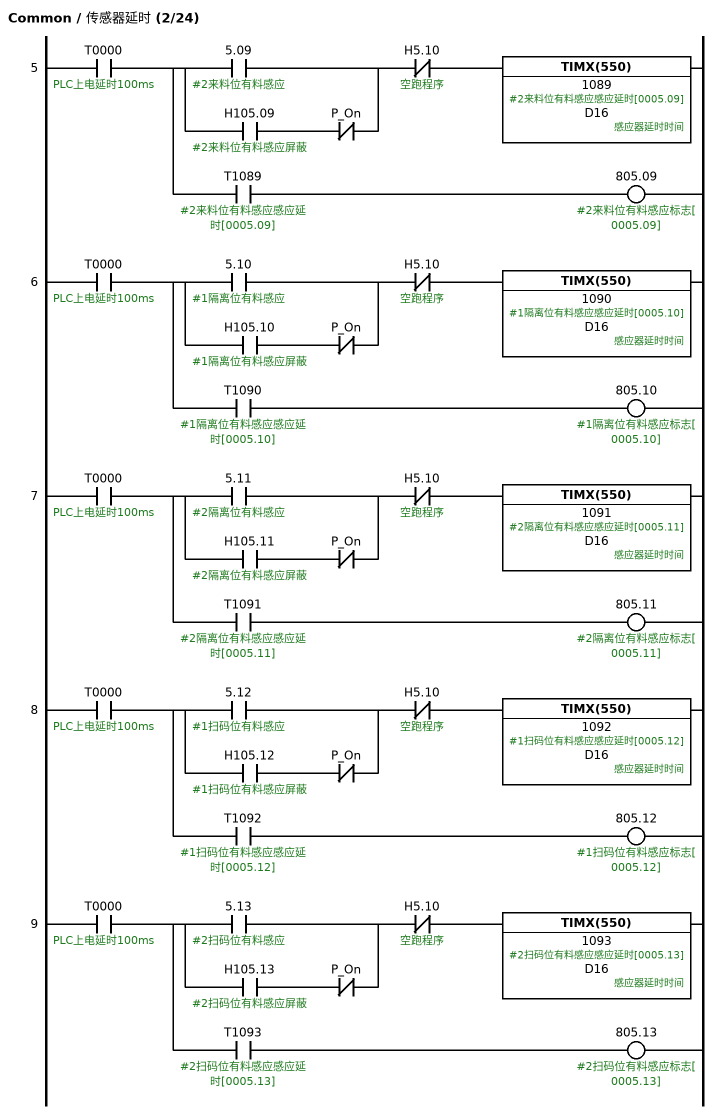
; [picture p504: Common / 传感器延时, rungs 5-9]
; rung 5
LD T0000  ; PLC上电延时100ms
OUT TR0
LD 5.09  ; #2来料位有料感应
LD H105.09  ; #2来料位有料感应屏蔽
ANDNOT P_On
ORLD
ANDLD
ANDNOT H5.10  ; 空跑程序
TIMX(550) 1089 D16  ; 感应器延时时间, #2来料位有料感应感应延时[0005.09]
LD TR0
AND T1089  ; #2来料位有料感应感应延时[0005.09]
OUT 805.09  ; #2来料位有料感应标志[0005.09]
; rung 6
LD T0000  ; PLC上电延时100ms
OUT TR0
LD 5.10  ; #1隔离位有料感应
LD H105.10  ; #1隔离位有料感应屏蔽
ANDNOT P_On
ORLD
ANDLD
ANDNOT H5.10  ; 空跑程序
TIMX(550) 1090 D16  ; 感应器延时时间, #1隔离位有料感应感应延时[0005.10]
LD TR0
AND T1090  ; #1隔离位有料感应感应延时[0005.10]
OUT 805.10  ; #1隔离位有料感应标志[0005.10]
; rung 7
LD T0000  ; PLC上电延时100ms
OUT TR0
LD 5.11  ; #2隔离位有料感应
LD H105.11  ; #2隔离位有料感应屏蔽
ANDNOT P_On
ORLD
ANDLD
ANDNOT H5.10  ; 空跑程序
TIMX(550) 1091 D16  ; 感应器延时时间, #2隔离位有料感应感应延时[0005.11]
LD TR0
AND T1091  ; #2隔离位有料感应感应延时[0005.11]
OUT 805.11  ; #2隔离位有料感应标志[0005.11]
; rung 8
LD T0000  ; PLC上电延时100ms
OUT TR0
LD 5.12  ; #1扫码位有料感应
LD H105.12  ; #1扫码位有料感应屏蔽
ANDNOT P_On
ORLD
ANDLD
ANDNOT H5.10  ; 空跑程序
TIMX(550) 1092 D16  ; 感应器延时时间, #1扫码位有料感应感应延时[0005.12]
LD TR0
AND T1092  ; #1扫码位有料感应感应延时[0005.12]
OUT 805.12  ; #1扫码位有料感应标志[0005.12]
; rung 9
LD T0000  ; PLC上电延时100ms
OUT TR0
LD 5.13  ; #2扫码位有料感应
LD H105.13  ; #2扫码位有料感应屏蔽
ANDNOT P_On
ORLD
ANDLD
ANDNOT H5.10  ; 空跑程序
TIMX(550) 1093 D16  ; 感应器延时时间, #2扫码位有料感应感应延时[0005.13]
LD TR0
AND T1093  ; #2扫码位有料感应感应延时[0005.13]
OUT 805.13  ; #2扫码位有料感应标志[0005.13]

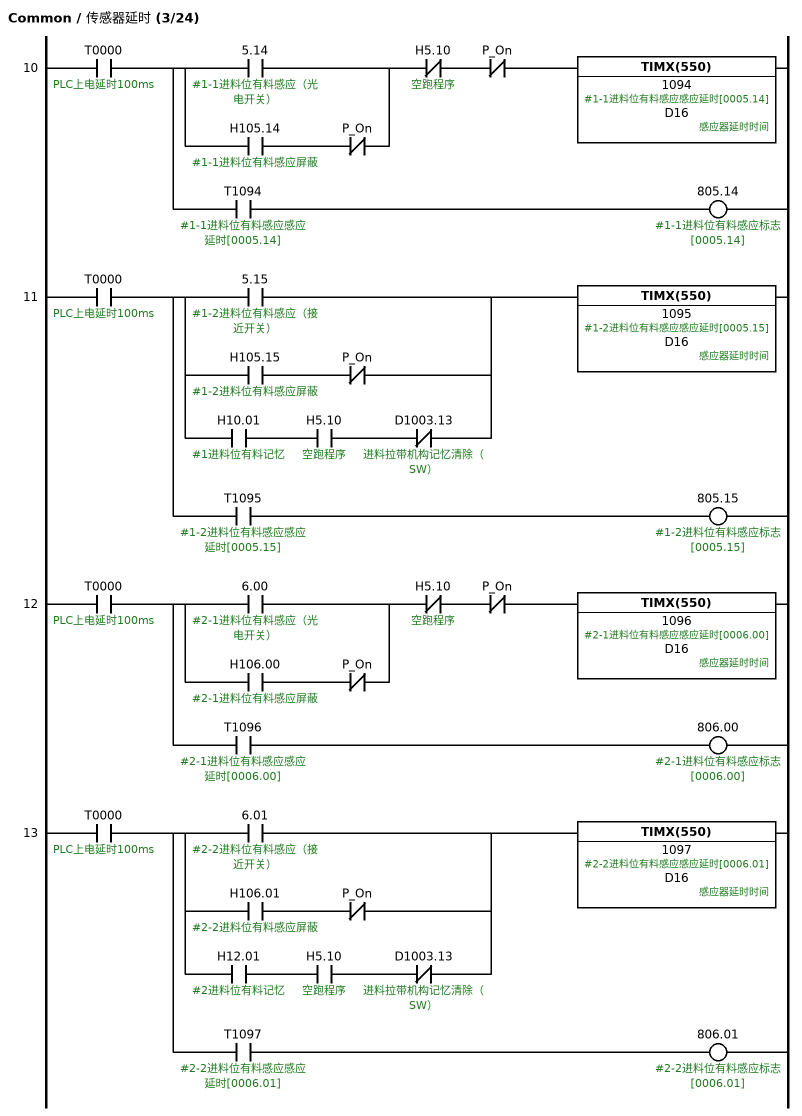
; rung 10
LD T0000  ; PLC上电延时100ms
OUT TR0
LD 5.14  ; #1-1进料位有料感应（光电开关）
LD H105.14  ; #1-1进料位有料感应屏蔽
ANDNOT P_On
ORLD
ANDLD
ANDNOT H5.10  ; 空跑程序
ANDNOT P_On
TIMX(550) 1094 D16  ; 感应器延时时间, #1-1进料位有料感应感应延时[0005.14]
LD TR0
AND T1094  ; #1-1进料位有料感应感应延时[0005.14]
OUT 805.14  ; #1-1进料位有料感应标志[0005.14]
; rung 11
LD T0000  ; PLC上电延时100ms
OUT TR0
LD 5.15  ; #1-2进料位有料感应（接近开关）
LD H105.15  ; #1-2进料位有料感应屏蔽
ANDNOT P_On
ORLD
LD H10.01  ; #1进料位有料记忆
AND H5.10  ; 空跑程序
ANDNOT D1003.13  ; 进料拉带机构记忆清除（SW）
ORLD
ANDLD
TIMX(550) 1095 D16  ; 感应器延时时间, #1-2进料位有料感应感应延时[0005.15]
LD TR0
AND T1095  ; #1-2进料位有料感应感应延时[0005.15]
OUT 805.15  ; #1-2进料位有料感应标志[0005.15]
; rung 12
LD T0000  ; PLC上电延时100ms
OUT TR0
LD 6.00  ; #2-1进料位有料感应（光电开关）
LD H106.00  ; #2-1进料位有料感应屏蔽
ANDNOT P_On
ORLD
ANDLD
ANDNOT H5.10  ; 空跑程序
ANDNOT P_On
TIMX(550) 1096 D16  ; 感应器延时时间, #2-1进料位有料感应感应延时[0006.00]
LD TR0
AND T1096  ; #2-1进料位有料感应感应延时[0006.00]
OUT 806.00  ; #2-1进料位有料感应标志[0006.00]
; rung 13
LD T0000  ; PLC上电延时100ms
OUT TR0
LD 6.01  ; #2-2进料位有料感应（接近开关）
LD H106.01  ; #2-2进料位有料感应屏蔽
ANDNOT P_On
ORLD
LD H12.01  ; #2进料位有料记忆
AND H5.10  ; 空跑程序
ANDNOT D1003.13  ; 进料拉带机构记忆清除（SW）
ORLD
ANDLD
TIMX(550) 1097 D16  ; 感应器延时时间, #2-2进料位有料感应感应延时[0006.01]
LD TR0
AND T1097  ; #2-2进料位有料感应感应延时[0006.01]
OUT 806.01  ; #2-2进料位有料感应标志[0006.01]

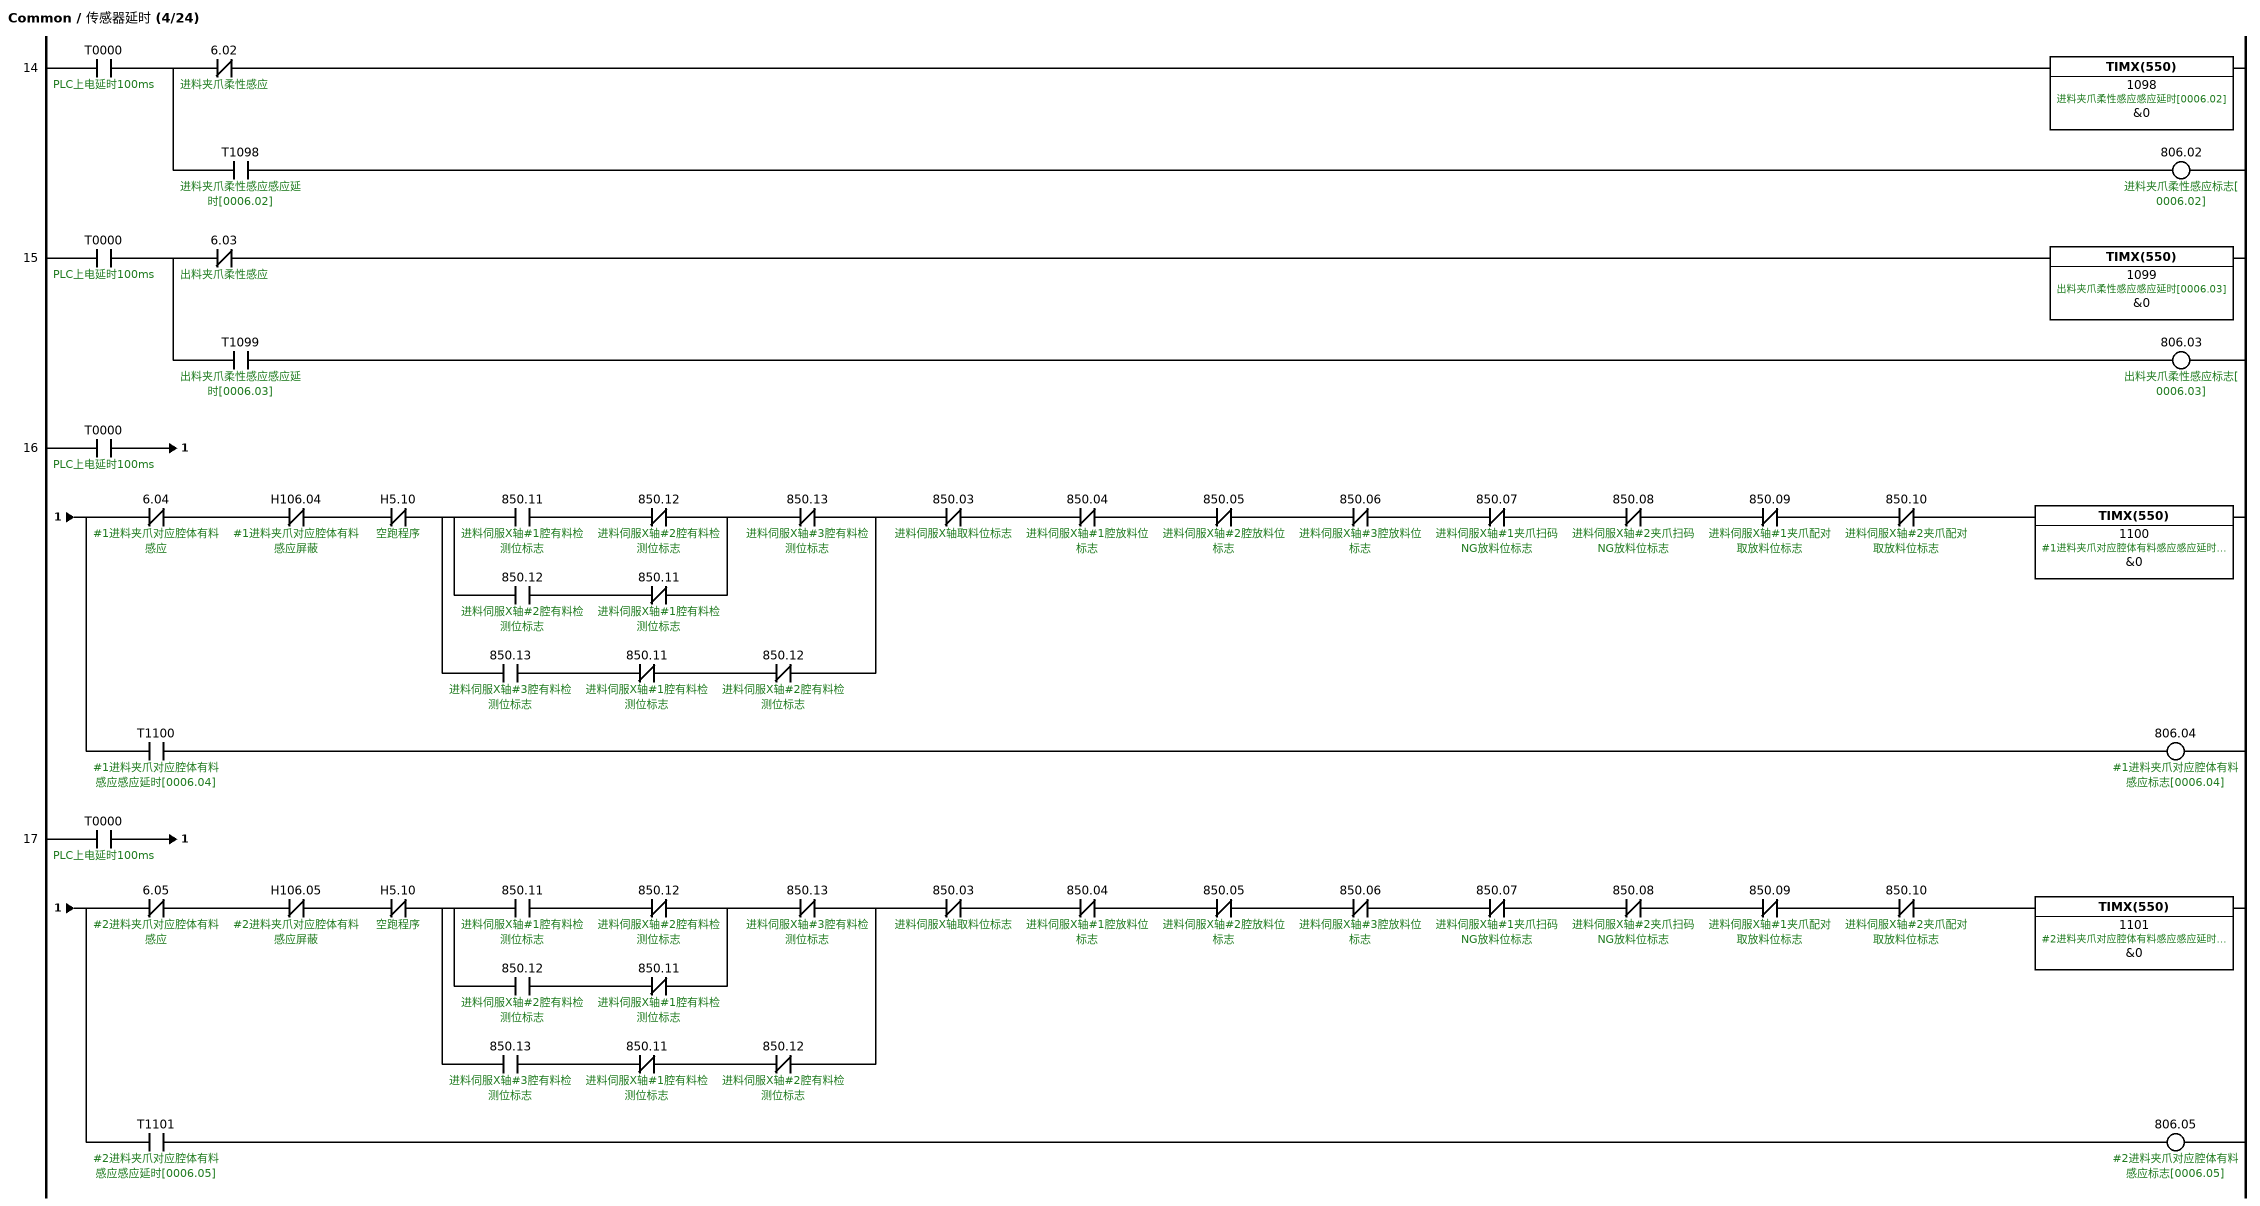
; rung 14
LD T0000  ; PLC上电延时100ms
OUT TR0
ANDNOT 6.02  ; 进料夹爪柔性感应
TIMX(550) 1098 &0  ; 进料夹爪柔性感应感应延时[0006.02]
LD TR0
AND T1098  ; 进料夹爪柔性感应感应延时[0006.02]
OUT 806.02  ; 进料夹爪柔性感应标志[0006.02]
; rung 15
LD T0000  ; PLC上电延时100ms
OUT TR0
ANDNOT 6.03  ; 出料夹爪柔性感应
TIMX(550) 1099 &0  ; 出料夹爪柔性感应感应延时[0006.03]
LD TR0
AND T1099  ; 出料夹爪柔性感应感应延时[0006.03]
OUT 806.03  ; 出料夹爪柔性感应标志[0006.03]
; rung 16
LD T0000  ; PLC上电延时100ms
OUT TR0
ANDNOT 6.04  ; #1进料夹爪对应腔体有料感应
ANDNOT H106.04  ; #1进料夹爪对应腔体有料感应屏蔽
ANDNOT H5.10  ; 空跑程序
LD 850.11  ; 进料伺服X轴#1腔有料检测位标志
ANDNOT 850.12  ; 进料伺服X轴#2腔有料检测位标志
LD 850.12  ; 进料伺服X轴#2腔有料检测位标志
ANDNOT 850.11  ; 进料伺服X轴#1腔有料检测位标志
ORLD
ANDNOT 850.13  ; 进料伺服X轴#3腔有料检测位标志
LD 850.13  ; 进料伺服X轴#3腔有料检测位标志
ANDNOT 850.11  ; 进料伺服X轴#1腔有料检测位标志
ANDNOT 850.12  ; 进料伺服X轴#2腔有料检测位标志
ORLD
ANDLD
ANDNOT 850.03  ; 进料伺服X轴取料位标志
ANDNOT 850.04  ; 进料伺服X轴#1腔放料位标志
ANDNOT 850.05  ; 进料伺服X轴#2腔放料位标志
ANDNOT 850.06  ; 进料伺服X轴#3腔放料位标志
ANDNOT 850.07  ; 进料伺服X轴#1夹爪扫码NG放料位标志
ANDNOT 850.08  ; 进料伺服X轴#2夹爪扫码NG放料位标志
ANDNOT 850.09  ; 进料伺服X轴#1夹爪配对取放料位标志
ANDNOT 850.10  ; 进料伺服X轴#2夹爪配对取放料位标志
TIMX(550) 1100 &0  ; #1进料夹爪对应腔体有料感应感应延时[0006.04]
LD TR0
AND T1100  ; #1进料夹爪对应腔体有料感应感应延时[0006.04]
OUT 806.04  ; #1进料夹爪对应腔体有料感应标志[0006.04]
; rung 17
LD T0000  ; PLC上电延时100ms
OUT TR0
ANDNOT 6.05  ; #2进料夹爪对应腔体有料感应
ANDNOT H106.05  ; #2进料夹爪对应腔体有料感应屏蔽
ANDNOT H5.10  ; 空跑程序
LD 850.11  ; 进料伺服X轴#1腔有料检测位标志
ANDNOT 850.12  ; 进料伺服X轴#2腔有料检测位标志
LD 850.12  ; 进料伺服X轴#2腔有料检测位标志
ANDNOT 850.11  ; 进料伺服X轴#1腔有料检测位标志
ORLD
ANDNOT 850.13  ; 进料伺服X轴#3腔有料检测位标志
LD 850.13  ; 进料伺服X轴#3腔有料检测位标志
ANDNOT 850.11  ; 进料伺服X轴#1腔有料检测位标志
ANDNOT 850.12  ; 进料伺服X轴#2腔有料检测位标志
ORLD
ANDLD
ANDNOT 850.03  ; 进料伺服X轴取料位标志
ANDNOT 850.04  ; 进料伺服X轴#1腔放料位标志
ANDNOT 850.05  ; 进料伺服X轴#2腔放料位标志
ANDNOT 850.06  ; 进料伺服X轴#3腔放料位标志
ANDNOT 850.07  ; 进料伺服X轴#1夹爪扫码NG放料位标志
ANDNOT 850.08  ; 进料伺服X轴#2夹爪扫码NG放料位标志
ANDNOT 850.09  ; 进料伺服X轴#1夹爪配对取放料位标志
ANDNOT 850.10  ; 进料伺服X轴#2夹爪配对取放料位标志
TIMX(550) 1101 &0  ; #2进料夹爪对应腔体有料感应感应延时[0006.05]
LD TR0
AND T1101  ; #2进料夹爪对应腔体有料感应感应延时[0006.05]
OUT 806.05  ; #2进料夹爪对应腔体有料感应标志[0006.05]

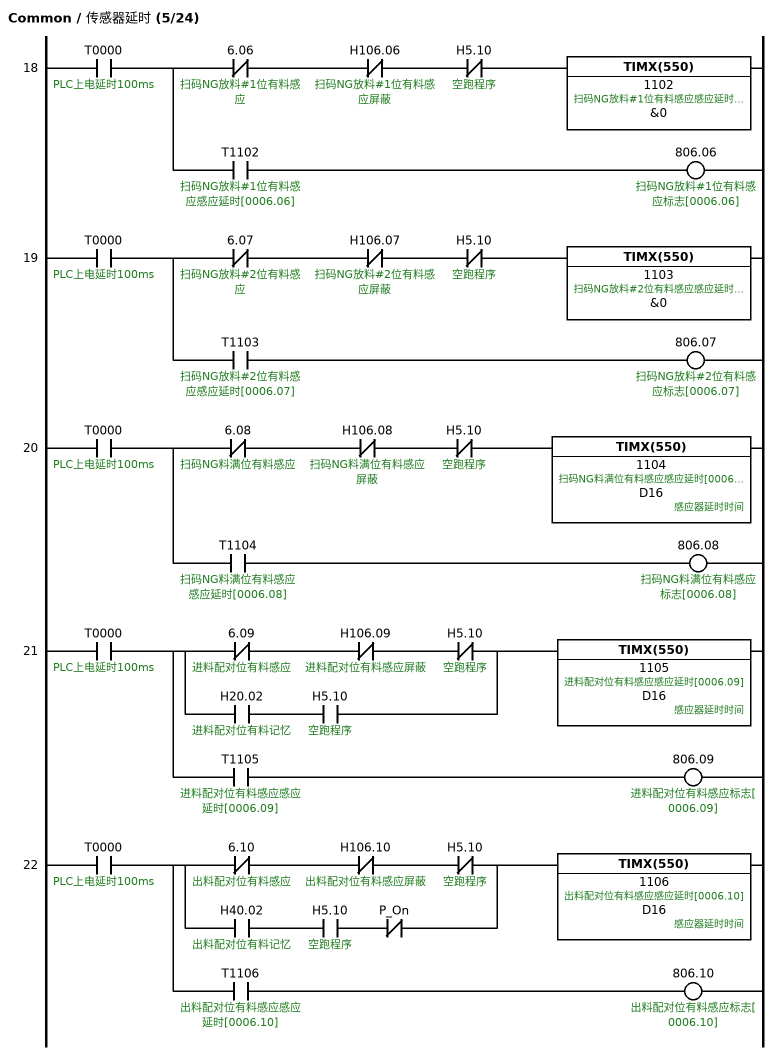
; rung 18
LD T0000  ; PLC上电延时100ms
OUT TR0
ANDNOT 6.06  ; 扫码NG放料#1位有料感应
ANDNOT H106.06  ; 扫码NG放料#1位有料感应屏蔽
ANDNOT H5.10  ; 空跑程序
TIMX(550) 1102 &0  ; 扫码NG放料#1位有料感应感应延时[0006.06]
LD TR0
AND T1102  ; 扫码NG放料#1位有料感应感应延时[0006.06]
OUT 806.06  ; 扫码NG放料#1位有料感应标志[0006.06]
; rung 19
LD T0000  ; PLC上电延时100ms
OUT TR0
ANDNOT 6.07  ; 扫码NG放料#2位有料感应
ANDNOT H106.07  ; 扫码NG放料#2位有料感应屏蔽
ANDNOT H5.10  ; 空跑程序
TIMX(550) 1103 &0  ; 扫码NG放料#2位有料感应感应延时[0006.07]
LD TR0
AND T1103  ; 扫码NG放料#2位有料感应感应延时[0006.07]
OUT 806.07  ; 扫码NG放料#2位有料感应标志[0006.07]
; rung 20
LD T0000  ; PLC上电延时100ms
OUT TR0
ANDNOT 6.08  ; 扫码NG料满位有料感应
ANDNOT H106.08  ; 扫码NG料满位有料感应屏蔽
ANDNOT H5.10  ; 空跑程序
TIMX(550) 1104 D16  ; 感应器延时时间, 扫码NG料满位有料感应感应延时[0006.08]
LD TR0
AND T1104  ; 扫码NG料满位有料感应感应延时[0006.08]
OUT 806.08  ; 扫码NG料满位有料感应标志[0006.08]
; rung 21
LD T0000  ; PLC上电延时100ms
OUT TR0
LDNOT 6.09  ; 进料配对位有料感应
ANDNOT H106.09  ; 进料配对位有料感应屏蔽
ANDNOT H5.10  ; 空跑程序
LD H20.02  ; 进料配对位有料记忆
AND H5.10  ; 空跑程序
ORLD
ANDLD
TIMX(550) 1105 D16  ; 感应器延时时间, 进料配对位有料感应感应延时[0006.09]
LD TR0
AND T1105  ; 进料配对位有料感应感应延时[0006.09]
OUT 806.09  ; 进料配对位有料感应标志[0006.09]
; rung 22
LD T0000  ; PLC上电延时100ms
OUT TR0
LDNOT 6.10  ; 出料配对位有料感应
ANDNOT H106.10  ; 出料配对位有料感应屏蔽
ANDNOT H5.10  ; 空跑程序
LD H40.02  ; 出料配对位有料记忆
AND H5.10  ; 空跑程序
ANDNOT P_On
ORLD
ANDLD
TIMX(550) 1106 D16  ; 感应器延时时间, 出料配对位有料感应感应延时[0006.10]
LD TR0
AND T1106  ; 出料配对位有料感应感应延时[0006.10]
OUT 806.10  ; 出料配对位有料感应标志[0006.10]

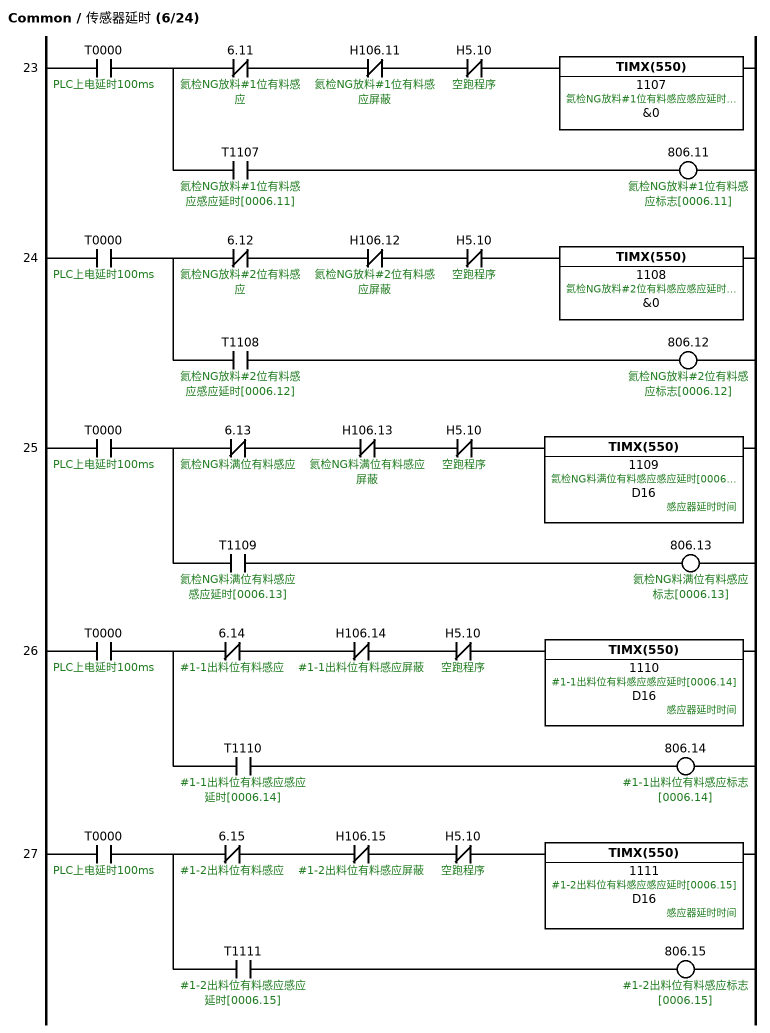
; rung 23
LD T0000  ; PLC上电延时100ms
OUT TR0
ANDNOT 6.11  ; 氦检NG放料#1位有料感应
ANDNOT H106.11  ; 氦检NG放料#1位有料感应屏蔽
ANDNOT H5.10  ; 空跑程序
TIMX(550) 1107 &0  ; 氦检NG放料#1位有料感应感应延时[0006.11]
LD TR0
AND T1107  ; 氦检NG放料#1位有料感应感应延时[0006.11]
OUT 806.11  ; 氦检NG放料#1位有料感应标志[0006.11]
; rung 24
LD T0000  ; PLC上电延时100ms
OUT TR0
ANDNOT 6.12  ; 氦检NG放料#2位有料感应
ANDNOT H106.12  ; 氦检NG放料#2位有料感应屏蔽
ANDNOT H5.10  ; 空跑程序
TIMX(550) 1108 &0  ; 氦检NG放料#2位有料感应感应延时[0006.12]
LD TR0
AND T1108  ; 氦检NG放料#2位有料感应感应延时[0006.12]
OUT 806.12  ; 氦检NG放料#2位有料感应标志[0006.12]
; rung 25
LD T0000  ; PLC上电延时100ms
OUT TR0
ANDNOT 6.13  ; 氦检NG料满位有料感应
ANDNOT H106.13  ; 氦检NG料满位有料感应屏蔽
ANDNOT H5.10  ; 空跑程序
TIMX(550) 1109 D16  ; 感应器延时时间, 氦检NG料满位有料感应感应延时[0006.13]
LD TR0
AND T1109  ; 氦检NG料满位有料感应感应延时[0006.13]
OUT 806.13  ; 氦检NG料满位有料感应标志[0006.13]
; rung 26
LD T0000  ; PLC上电延时100ms
OUT TR0
ANDNOT 6.14  ; #1-1出料位有料感应
ANDNOT H106.14  ; #1-1出料位有料感应屏蔽
ANDNOT H5.10  ; 空跑程序
TIMX(550) 1110 D16  ; 感应器延时时间, #1-1出料位有料感应感应延时[0006.14]
LD TR0
AND T1110  ; #1-1出料位有料感应感应延时[0006.14]
OUT 806.14  ; #1-1出料位有料感应标志[0006.14]
; rung 27
LD T0000  ; PLC上电延时100ms
OUT TR0
ANDNOT 6.15  ; #1-2出料位有料感应
ANDNOT H106.15  ; #1-2出料位有料感应屏蔽
ANDNOT H5.10  ; 空跑程序
TIMX(550) 1111 D16  ; 感应器延时时间, #1-2出料位有料感应感应延时[0006.15]
LD TR0
AND T1111  ; #1-2出料位有料感应感应延时[0006.15]
OUT 806.15  ; #1-2出料位有料感应标志[0006.15]

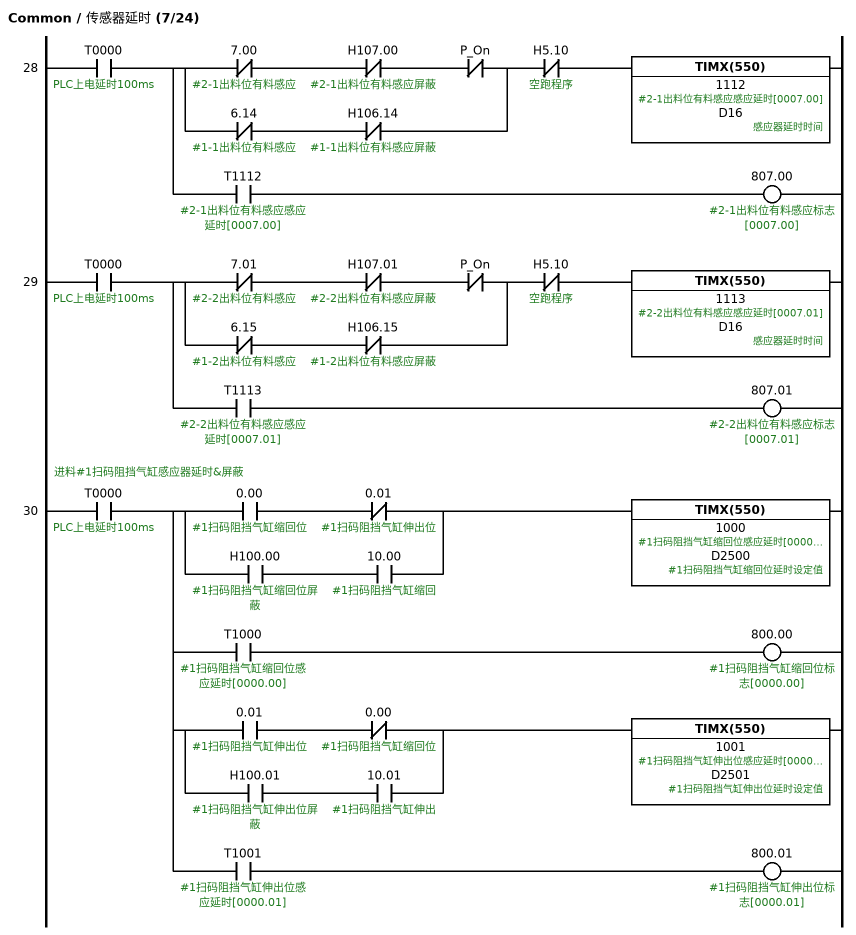
; rung 28
LD T0000  ; PLC上电延时100ms
OUT TR0
LDNOT 7.00  ; #2-1出料位有料感应
ANDNOT H107.00  ; #2-1出料位有料感应屏蔽
ANDNOT P_On
LDNOT 6.14  ; #1-1出料位有料感应
ANDNOT H106.14  ; #1-1出料位有料感应屏蔽
ORLD
ANDLD
ANDNOT H5.10  ; 空跑程序
TIMX(550) 1112 D16  ; 感应器延时时间, #2-1出料位有料感应感应延时[0007.00]
LD TR0
AND T1112  ; #2-1出料位有料感应感应延时[0007.00]
OUT 807.00  ; #2-1出料位有料感应标志[0007.00]
; rung 29
LD T0000  ; PLC上电延时100ms
OUT TR0
LDNOT 7.01  ; #2-2出料位有料感应
ANDNOT H107.01  ; #2-2出料位有料感应屏蔽
ANDNOT P_On
LDNOT 6.15  ; #1-2出料位有料感应
ANDNOT H106.15  ; #1-2出料位有料感应屏蔽
ORLD
ANDLD
ANDNOT H5.10  ; 空跑程序
TIMX(550) 1113 D16  ; 感应器延时时间, #2-2出料位有料感应感应延时[0007.01]
LD TR0
AND T1113  ; #2-2出料位有料感应感应延时[0007.01]
OUT 807.01  ; #2-2出料位有料感应标志[0007.01]
; rung 30: 进料#1扫码阻挡气缸感应器延时&屏蔽
LD T0000  ; PLC上电延时100ms
OUT TR0
LD 0.00  ; #1扫码阻挡气缸缩回位
ANDNOT 0.01  ; #1扫码阻挡气缸伸出位
LD H100.00  ; #1扫码阻挡气缸缩回位屏蔽
AND 10.00  ; #1扫码阻挡气缸缩回
ORLD
ANDLD
TIMX(550) 1000 D2500  ; #1扫码阻挡气缸缩回位延时设定值, #1扫码阻挡气缸缩回位感应延时[0000.00]
LD TR0
AND T1000  ; #1扫码阻挡气缸缩回位感应延时[0000.00]
OUT 800.00  ; #1扫码阻挡气缸缩回位标志[0000.00]
LD TR0
LD 0.01  ; #1扫码阻挡气缸伸出位
ANDNOT 0.00  ; #1扫码阻挡气缸缩回位
LD H100.01  ; #1扫码阻挡气缸伸出位屏蔽
AND 10.01  ; #1扫码阻挡气缸伸出
ORLD
ANDLD
TIMX(550) 1001 D2501  ; #1扫码阻挡气缸伸出位延时设定值, #1扫码阻挡气缸伸出位感应延时[0000.01]
LD TR0
AND T1001  ; #1扫码阻挡气缸伸出位感应延时[0000.01]
OUT 800.01  ; #1扫码阻挡气缸伸出位标志[0000.01]

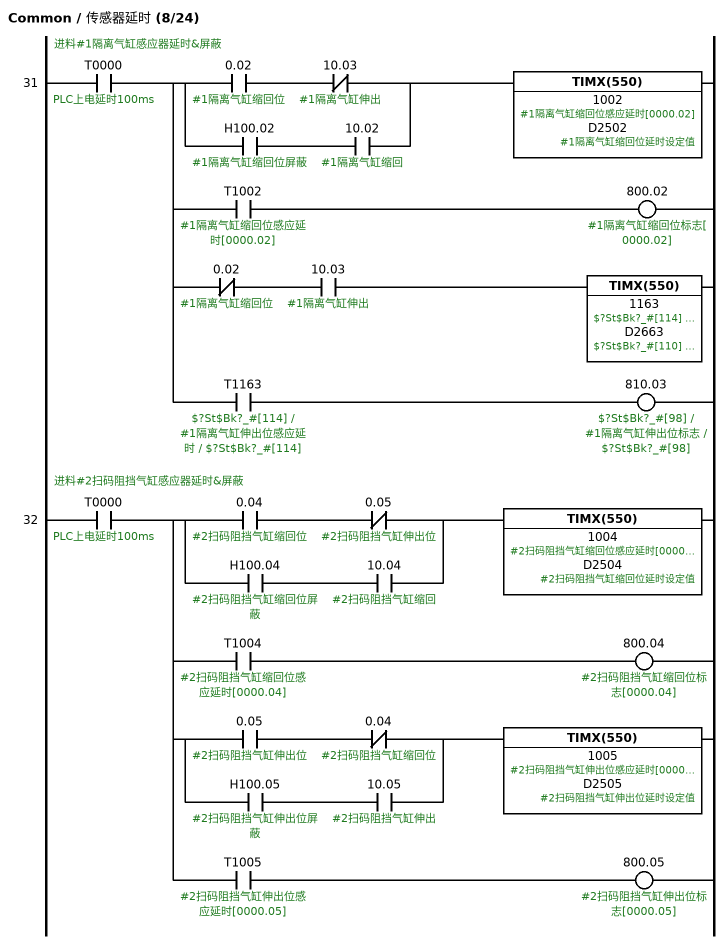
; rung 31: 进料#1隔离气缸感应器延时&屏蔽
LD T0000  ; PLC上电延时100ms
OUT TR0
LD 0.02  ; #1隔离气缸缩回位
ANDNOT 10.03  ; #1隔离气缸伸出
LD H100.02  ; #1隔离气缸缩回位屏蔽
AND 10.02  ; #1隔离气缸缩回
ORLD
ANDLD
TIMX(550) 1002 D2502  ; #1隔离气缸缩回位延时设定值, #1隔离气缸缩回位感应延时[0000.02]
LD TR0
AND T1002  ; #1隔离气缸缩回位感应延时[0000.02]
OUT 800.02  ; #1隔离气缸缩回位标志[0000.02]
LD TR0
ANDNOT 0.02  ; #1隔离气缸缩回位
AND 10.03  ; #1隔离气缸伸出
TIMX(550) 1163 D2663  ; $?St$Bk?_#[110] / #1隔离气缸伸出位延时设定值 / $?St$Bk?_#[110], $?St$Bk?_#[114] / #1隔离气缸伸出位感应延时 / $?St$Bk?_#[114]
LD TR0
AND T1163  ; $?St$Bk?_#[114] / #1隔离气缸伸出位感应延时 / $?St$Bk?_#[114]
OUT 810.03  ; $?St$Bk?_#[98] / #1隔离气缸伸出位标志 / $?St$Bk?_#[98]
; rung 32: 进料#2扫码阻挡气缸感应器延时&屏蔽
LD T0000  ; PLC上电延时100ms
OUT TR0
LD 0.04  ; #2扫码阻挡气缸缩回位
ANDNOT 0.05  ; #2扫码阻挡气缸伸出位
LD H100.04  ; #2扫码阻挡气缸缩回位屏蔽
AND 10.04  ; #2扫码阻挡气缸缩回
ORLD
ANDLD
TIMX(550) 1004 D2504  ; #2扫码阻挡气缸缩回位延时设定值, #2扫码阻挡气缸缩回位感应延时[0000.04]
LD TR0
AND T1004  ; #2扫码阻挡气缸缩回位感应延时[0000.04]
OUT 800.04  ; #2扫码阻挡气缸缩回位标志[0000.04]
LD TR0
LD 0.05  ; #2扫码阻挡气缸伸出位
ANDNOT 0.04  ; #2扫码阻挡气缸缩回位
LD H100.05  ; #2扫码阻挡气缸伸出位屏蔽
AND 10.05  ; #2扫码阻挡气缸伸出
ORLD
ANDLD
TIMX(550) 1005 D2505  ; #2扫码阻挡气缸伸出位延时设定值, #2扫码阻挡气缸伸出位感应延时[0000.05]
LD TR0
AND T1005  ; #2扫码阻挡气缸伸出位感应延时[0000.05]
OUT 800.05  ; #2扫码阻挡气缸伸出位标志[0000.05]

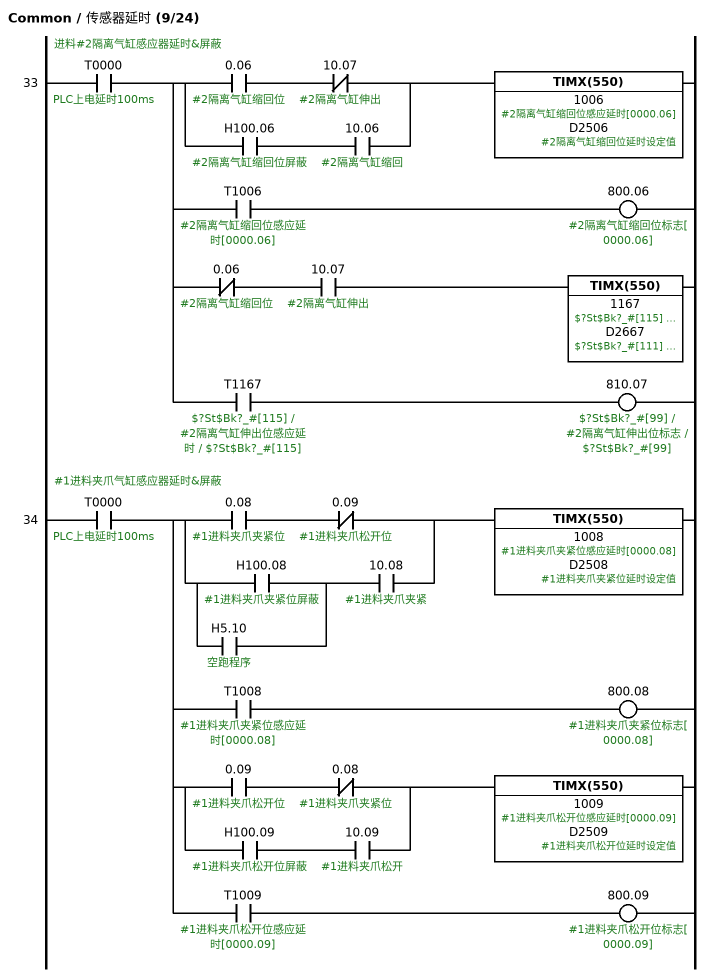
; rung 33: 进料#2隔离气缸感应器延时&屏蔽
LD T0000  ; PLC上电延时100ms
OUT TR0
LD 0.06  ; #2隔离气缸缩回位
ANDNOT 10.07  ; #2隔离气缸伸出
LD H100.06  ; #2隔离气缸缩回位屏蔽
AND 10.06  ; #2隔离气缸缩回
ORLD
ANDLD
TIMX(550) 1006 D2506  ; #2隔离气缸缩回位延时设定值, #2隔离气缸缩回位感应延时[0000.06]
LD TR0
AND T1006  ; #2隔离气缸缩回位感应延时[0000.06]
OUT 800.06  ; #2隔离气缸缩回位标志[0000.06]
LD TR0
ANDNOT 0.06  ; #2隔离气缸缩回位
AND 10.07  ; #2隔离气缸伸出
TIMX(550) 1167 D2667  ; $?St$Bk?_#[111] / #2隔离气缸伸出位延时设定值 / $?St$Bk?_#[111], $?St$Bk?_#[115] / #2隔离气缸伸出位感应延时 / $?St$Bk?_#[115]
LD TR0
AND T1167  ; $?St$Bk?_#[115] / #2隔离气缸伸出位感应延时 / $?St$Bk?_#[115]
OUT 810.07  ; $?St$Bk?_#[99] / #2隔离气缸伸出位标志 / $?St$Bk?_#[99]
; rung 34: #1进料夹爪气缸感应器延时&屏蔽
LD T0000  ; PLC上电延时100ms
OUT TR0
LD 0.08  ; #1进料夹爪夹紧位
ANDNOT 0.09  ; #1进料夹爪松开位
LD H100.08  ; #1进料夹爪夹紧位屏蔽
OR H5.10  ; 空跑程序
AND 10.08  ; #1进料夹爪夹紧
ORLD
ANDLD
TIMX(550) 1008 D2508  ; #1进料夹爪夹紧位延时设定值, #1进料夹爪夹紧位感应延时[0000.08]
LD TR0
AND T1008  ; #1进料夹爪夹紧位感应延时[0000.08]
OUT 800.08  ; #1进料夹爪夹紧位标志[0000.08]
LD TR0
LD 0.09  ; #1进料夹爪松开位
ANDNOT 0.08  ; #1进料夹爪夹紧位
LD H100.09  ; #1进料夹爪松开位屏蔽
AND 10.09  ; #1进料夹爪松开
ORLD
ANDLD
TIMX(550) 1009 D2509  ; #1进料夹爪松开位延时设定值, #1进料夹爪松开位感应延时[0000.09]
LD TR0
AND T1009  ; #1进料夹爪松开位感应延时[0000.09]
OUT 800.09  ; #1进料夹爪松开位标志[0000.09]

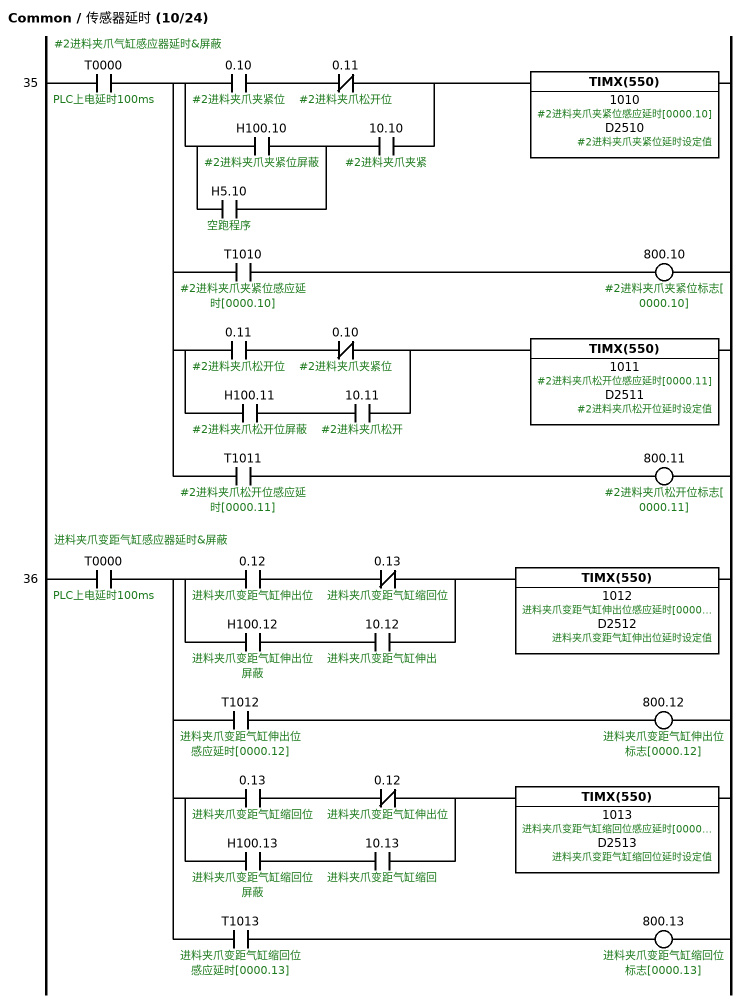
; rung 35: #2进料夹爪气缸感应器延时&屏蔽
LD T0000  ; PLC上电延时100ms
OUT TR0
LD 0.10  ; #2进料夹爪夹紧位
ANDNOT 0.11  ; #2进料夹爪松开位
LD H100.10  ; #2进料夹爪夹紧位屏蔽
OR H5.10  ; 空跑程序
AND 10.10  ; #2进料夹爪夹紧
ORLD
ANDLD
TIMX(550) 1010 D2510  ; #2进料夹爪夹紧位延时设定值, #2进料夹爪夹紧位感应延时[0000.10]
LD TR0
AND T1010  ; #2进料夹爪夹紧位感应延时[0000.10]
OUT 800.10  ; #2进料夹爪夹紧位标志[0000.10]
LD TR0
LD 0.11  ; #2进料夹爪松开位
ANDNOT 0.10  ; #2进料夹爪夹紧位
LD H100.11  ; #2进料夹爪松开位屏蔽
AND 10.11  ; #2进料夹爪松开
ORLD
ANDLD
TIMX(550) 1011 D2511  ; #2进料夹爪松开位延时设定值, #2进料夹爪松开位感应延时[0000.11]
LD TR0
AND T1011  ; #2进料夹爪松开位感应延时[0000.11]
OUT 800.11  ; #2进料夹爪松开位标志[0000.11]
; rung 36: 进料夹爪变距气缸感应器延时&屏蔽
LD T0000  ; PLC上电延时100ms
OUT TR0
LD 0.12  ; 进料夹爪变距气缸伸出位
ANDNOT 0.13  ; 进料夹爪变距气缸缩回位
LD H100.12  ; 进料夹爪变距气缸伸出位屏蔽
AND 10.12  ; 进料夹爪变距气缸伸出
ORLD
ANDLD
TIMX(550) 1012 D2512  ; 进料夹爪变距气缸伸出位延时设定值, 进料夹爪变距气缸伸出位感应延时[0000.12]
LD TR0
AND T1012  ; 进料夹爪变距气缸伸出位感应延时[0000.12]
OUT 800.12  ; 进料夹爪变距气缸伸出位标志[0000.12]
LD TR0
LD 0.13  ; 进料夹爪变距气缸缩回位
ANDNOT 0.12  ; 进料夹爪变距气缸伸出位
LD H100.13  ; 进料夹爪变距气缸缩回位屏蔽
AND 10.13  ; 进料夹爪变距气缸缩回
ORLD
ANDLD
TIMX(550) 1013 D2513  ; 进料夹爪变距气缸缩回位延时设定值, 进料夹爪变距气缸缩回位感应延时[0000.13]
LD TR0
AND T1013  ; 进料夹爪变距气缸缩回位感应延时[0000.13]
OUT 800.13  ; 进料夹爪变距气缸缩回位标志[0000.13]

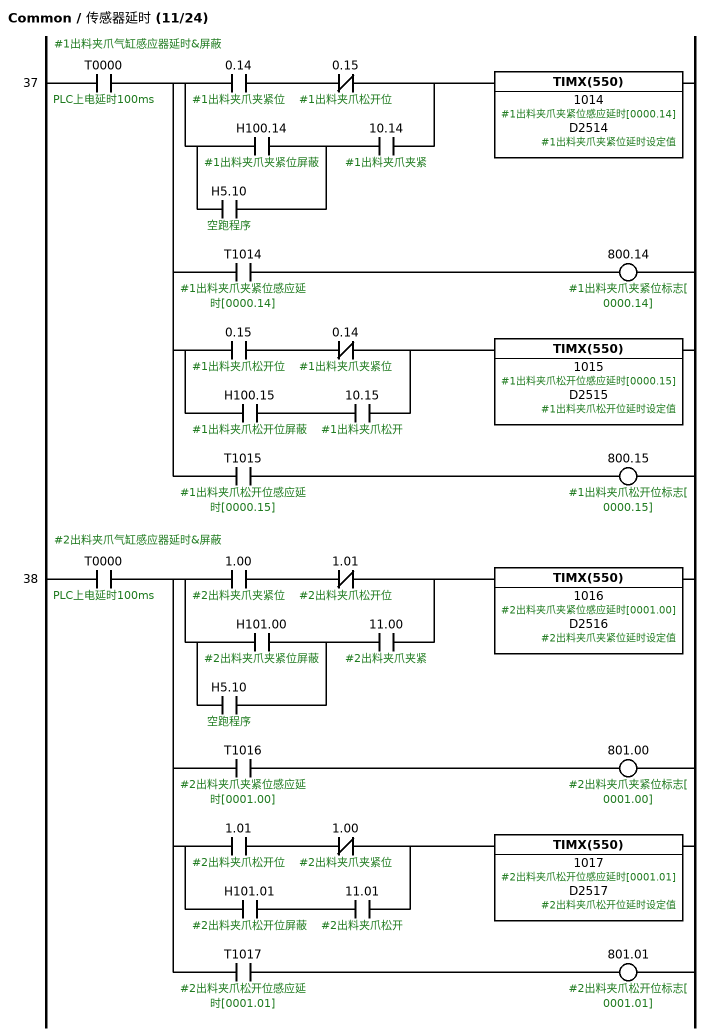
; rung 37: #1出料夹爪气缸感应器延时&屏蔽
LD T0000  ; PLC上电延时100ms
OUT TR0
LD 0.14  ; #1出料夹爪夹紧位
ANDNOT 0.15  ; #1出料夹爪松开位
LD H100.14  ; #1出料夹爪夹紧位屏蔽
OR H5.10  ; 空跑程序
AND 10.14  ; #1出料夹爪夹紧
ORLD
ANDLD
TIMX(550) 1014 D2514  ; #1出料夹爪夹紧位延时设定值, #1出料夹爪夹紧位感应延时[0000.14]
LD TR0
AND T1014  ; #1出料夹爪夹紧位感应延时[0000.14]
OUT 800.14  ; #1出料夹爪夹紧位标志[0000.14]
LD TR0
LD 0.15  ; #1出料夹爪松开位
ANDNOT 0.14  ; #1出料夹爪夹紧位
LD H100.15  ; #1出料夹爪松开位屏蔽
AND 10.15  ; #1出料夹爪松开
ORLD
ANDLD
TIMX(550) 1015 D2515  ; #1出料夹爪松开位延时设定值, #1出料夹爪松开位感应延时[0000.15]
LD TR0
AND T1015  ; #1出料夹爪松开位感应延时[0000.15]
OUT 800.15  ; #1出料夹爪松开位标志[0000.15]
; rung 38: #2出料夹爪气缸感应器延时&屏蔽
LD T0000  ; PLC上电延时100ms
OUT TR0
LD 1.00  ; #2出料夹爪夹紧位
ANDNOT 1.01  ; #2出料夹爪松开位
LD H101.00  ; #2出料夹爪夹紧位屏蔽
OR H5.10  ; 空跑程序
AND 11.00  ; #2出料夹爪夹紧
ORLD
ANDLD
TIMX(550) 1016 D2516  ; #2出料夹爪夹紧位延时设定值, #2出料夹爪夹紧位感应延时[0001.00]
LD TR0
AND T1016  ; #2出料夹爪夹紧位感应延时[0001.00]
OUT 801.00  ; #2出料夹爪夹紧位标志[0001.00]
LD TR0
LD 1.01  ; #2出料夹爪松开位
ANDNOT 1.00  ; #2出料夹爪夹紧位
LD H101.01  ; #2出料夹爪松开位屏蔽
AND 11.01  ; #2出料夹爪松开
ORLD
ANDLD
TIMX(550) 1017 D2517  ; #2出料夹爪松开位延时设定值, #2出料夹爪松开位感应延时[0001.01]
LD TR0
AND T1017  ; #2出料夹爪松开位感应延时[0001.01]
OUT 801.01  ; #2出料夹爪松开位标志[0001.01]

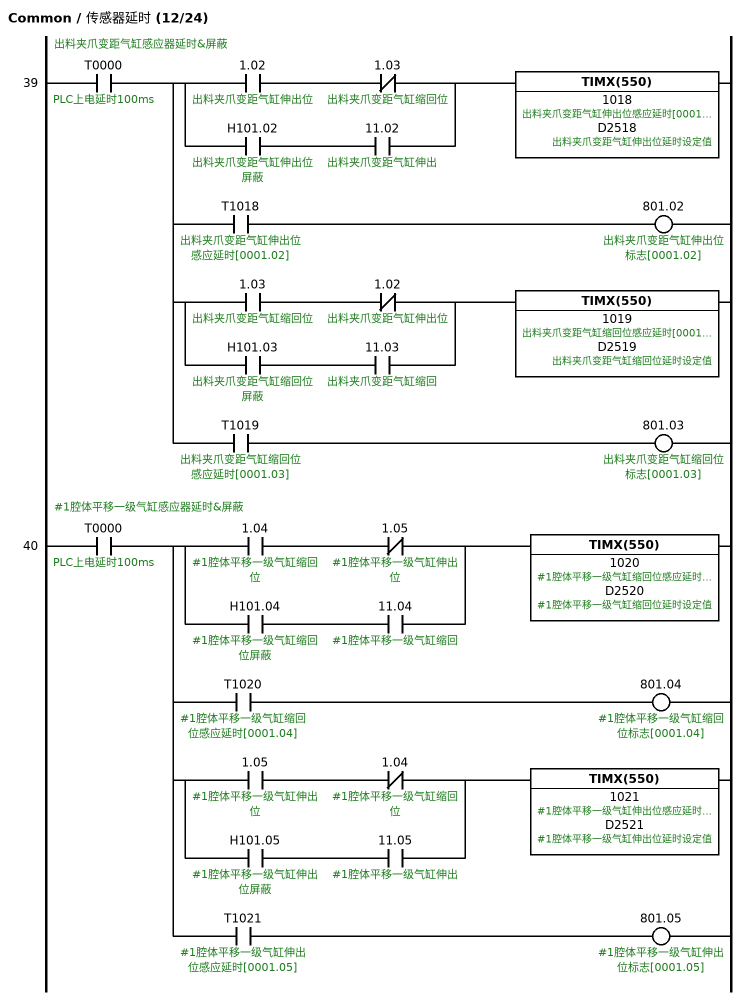
; rung 39: 出料夹爪变距气缸感应器延时&屏蔽
LD T0000  ; PLC上电延时100ms
OUT TR0
LD 1.02  ; 出料夹爪变距气缸伸出位
ANDNOT 1.03  ; 出料夹爪变距气缸缩回位
LD H101.02  ; 出料夹爪变距气缸伸出位屏蔽
AND 11.02  ; 出料夹爪变距气缸伸出
ORLD
ANDLD
TIMX(550) 1018 D2518  ; 出料夹爪变距气缸伸出位延时设定值, 出料夹爪变距气缸伸出位感应延时[0001.02]
LD TR0
AND T1018  ; 出料夹爪变距气缸伸出位感应延时[0001.02]
OUT 801.02  ; 出料夹爪变距气缸伸出位标志[0001.02]
LD TR0
LD 1.03  ; 出料夹爪变距气缸缩回位
ANDNOT 1.02  ; 出料夹爪变距气缸伸出位
LD H101.03  ; 出料夹爪变距气缸缩回位屏蔽
AND 11.03  ; 出料夹爪变距气缸缩回
ORLD
ANDLD
TIMX(550) 1019 D2519  ; 出料夹爪变距气缸缩回位延时设定值, 出料夹爪变距气缸缩回位感应延时[0001.03]
LD TR0
AND T1019  ; 出料夹爪变距气缸缩回位感应延时[0001.03]
OUT 801.03  ; 出料夹爪变距气缸缩回位标志[0001.03]
; rung 40: #1腔体平移一级气缸感应器延时&屏蔽
LD T0000  ; PLC上电延时100ms
OUT TR0
LD 1.04  ; #1腔体平移一级气缸缩回位
ANDNOT 1.05  ; #1腔体平移一级气缸伸出位
LD H101.04  ; #1腔体平移一级气缸缩回位屏蔽
AND 11.04  ; #1腔体平移一级气缸缩回
ORLD
ANDLD
TIMX(550) 1020 D2520  ; #1腔体平移一级气缸缩回位延时设定值, #1腔体平移一级气缸缩回位感应延时[0001.04]
LD TR0
AND T1020  ; #1腔体平移一级气缸缩回位感应延时[0001.04]
OUT 801.04  ; #1腔体平移一级气缸缩回位标志[0001.04]
LD TR0
LD 1.05  ; #1腔体平移一级气缸伸出位
ANDNOT 1.04  ; #1腔体平移一级气缸缩回位
LD H101.05  ; #1腔体平移一级气缸伸出位屏蔽
AND 11.05  ; #1腔体平移一级气缸伸出
ORLD
ANDLD
TIMX(550) 1021 D2521  ; #1腔体平移一级气缸伸出位延时设定值, #1腔体平移一级气缸伸出位感应延时[0001.05]
LD TR0
AND T1021  ; #1腔体平移一级气缸伸出位感应延时[0001.05]
OUT 801.05  ; #1腔体平移一级气缸伸出位标志[0001.05]

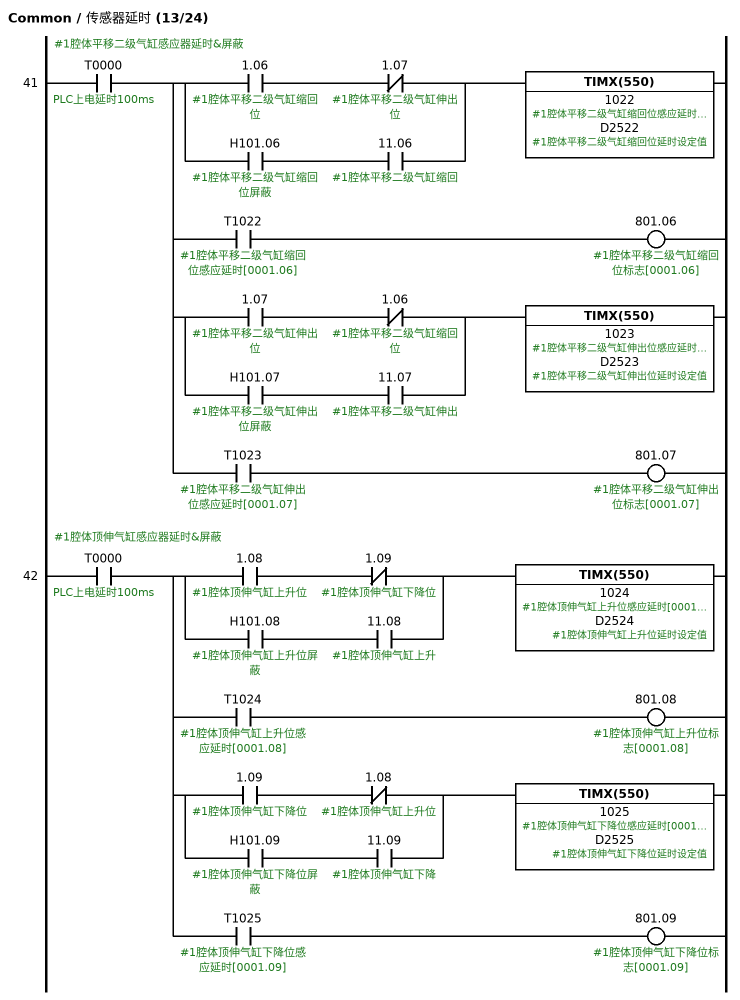
; rung 41: #1腔体平移二级气缸感应器延时&屏蔽
LD T0000  ; PLC上电延时100ms
OUT TR0
LD 1.06  ; #1腔体平移二级气缸缩回位
ANDNOT 1.07  ; #1腔体平移二级气缸伸出位
LD H101.06  ; #1腔体平移二级气缸缩回位屏蔽
AND 11.06  ; #1腔体平移二级气缸缩回
ORLD
ANDLD
TIMX(550) 1022 D2522  ; #1腔体平移二级气缸缩回位延时设定值, #1腔体平移二级气缸缩回位感应延时[0001.06]
LD TR0
AND T1022  ; #1腔体平移二级气缸缩回位感应延时[0001.06]
OUT 801.06  ; #1腔体平移二级气缸缩回位标志[0001.06]
LD TR0
LD 1.07  ; #1腔体平移二级气缸伸出位
ANDNOT 1.06  ; #1腔体平移二级气缸缩回位
LD H101.07  ; #1腔体平移二级气缸伸出位屏蔽
AND 11.07  ; #1腔体平移二级气缸伸出
ORLD
ANDLD
TIMX(550) 1023 D2523  ; #1腔体平移二级气缸伸出位延时设定值, #1腔体平移二级气缸伸出位感应延时[0001.07]
LD TR0
AND T1023  ; #1腔体平移二级气缸伸出位感应延时[0001.07]
OUT 801.07  ; #1腔体平移二级气缸伸出位标志[0001.07]
; rung 42: #1腔体顶伸气缸感应器延时&屏蔽
LD T0000  ; PLC上电延时100ms
OUT TR0
LD 1.08  ; #1腔体顶伸气缸上升位
ANDNOT 1.09  ; #1腔体顶伸气缸下降位
LD H101.08  ; #1腔体顶伸气缸上升位屏蔽
AND 11.08  ; #1腔体顶伸气缸上升
ORLD
ANDLD
TIMX(550) 1024 D2524  ; #1腔体顶伸气缸上升位延时设定值, #1腔体顶伸气缸上升位感应延时[0001.08]
LD TR0
AND T1024  ; #1腔体顶伸气缸上升位感应延时[0001.08]
OUT 801.08  ; #1腔体顶伸气缸上升位标志[0001.08]
LD TR0
LD 1.09  ; #1腔体顶伸气缸下降位
ANDNOT 1.08  ; #1腔体顶伸气缸上升位
LD H101.09  ; #1腔体顶伸气缸下降位屏蔽
AND 11.09  ; #1腔体顶伸气缸下降
ORLD
ANDLD
TIMX(550) 1025 D2525  ; #1腔体顶伸气缸下降位延时设定值, #1腔体顶伸气缸下降位感应延时[0001.09]
LD TR0
AND T1025  ; #1腔体顶伸气缸下降位感应延时[0001.09]
OUT 801.09  ; #1腔体顶伸气缸下降位标志[0001.09]

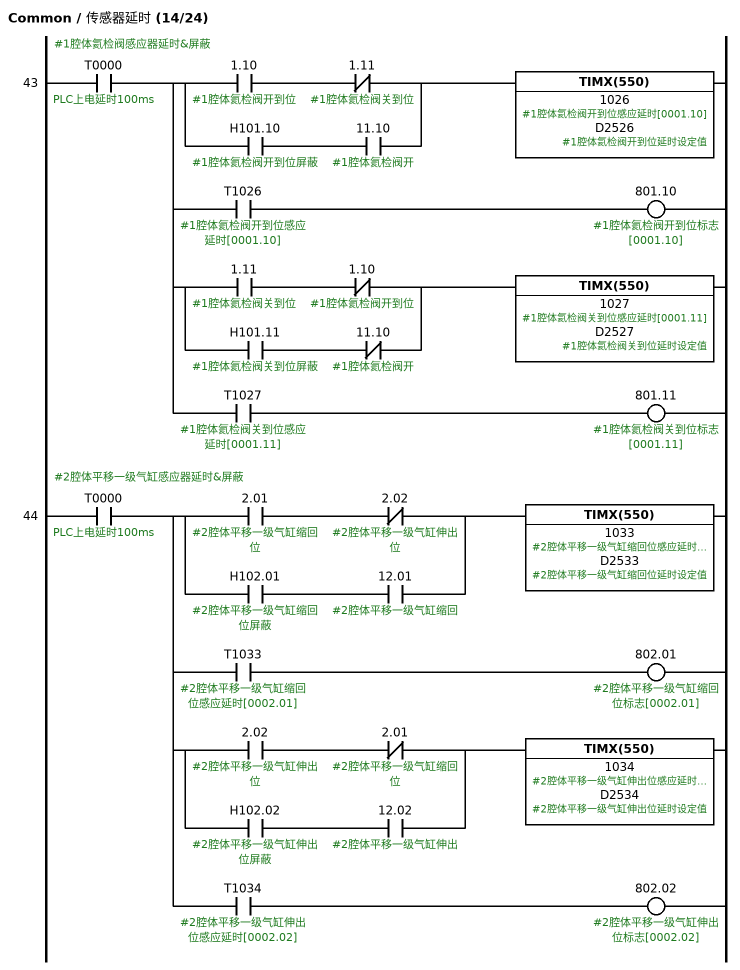
; rung 43: #1腔体氦检阀感应器延时&屏蔽
LD T0000  ; PLC上电延时100ms
OUT TR0
LD 1.10  ; #1腔体氦检阀开到位
ANDNOT 1.11  ; #1腔体氦检阀关到位
LD H101.10  ; #1腔体氦检阀开到位屏蔽
AND 11.10  ; #1腔体氦检阀开
ORLD
ANDLD
TIMX(550) 1026 D2526  ; #1腔体氦检阀开到位延时设定值, #1腔体氦检阀开到位感应延时[0001.10]
LD TR0
AND T1026  ; #1腔体氦检阀开到位感应延时[0001.10]
OUT 801.10  ; #1腔体氦检阀开到位标志[0001.10]
LD TR0
LD 1.11  ; #1腔体氦检阀关到位
ANDNOT 1.10  ; #1腔体氦检阀开到位
LD H101.11  ; #1腔体氦检阀关到位屏蔽
ANDNOT 11.10  ; #1腔体氦检阀开
ORLD
ANDLD
TIMX(550) 1027 D2527  ; #1腔体氦检阀关到位延时设定值, #1腔体氦检阀关到位感应延时[0001.11]
LD TR0
AND T1027  ; #1腔体氦检阀关到位感应延时[0001.11]
OUT 801.11  ; #1腔体氦检阀关到位标志[0001.11]
; rung 44: #2腔体平移一级气缸感应器延时&屏蔽
LD T0000  ; PLC上电延时100ms
OUT TR0
LD 2.01  ; #2腔体平移一级气缸缩回位
ANDNOT 2.02  ; #2腔体平移一级气缸伸出位
LD H102.01  ; #2腔体平移一级气缸缩回位屏蔽
AND 12.01  ; #2腔体平移一级气缸缩回
ORLD
ANDLD
TIMX(550) 1033 D2533  ; #2腔体平移一级气缸缩回位延时设定值, #2腔体平移一级气缸缩回位感应延时[0002.01]
LD TR0
AND T1033  ; #2腔体平移一级气缸缩回位感应延时[0002.01]
OUT 802.01  ; #2腔体平移一级气缸缩回位标志[0002.01]
LD TR0
LD 2.02  ; #2腔体平移一级气缸伸出位
ANDNOT 2.01  ; #2腔体平移一级气缸缩回位
LD H102.02  ; #2腔体平移一级气缸伸出位屏蔽
AND 12.02  ; #2腔体平移一级气缸伸出
ORLD
ANDLD
TIMX(550) 1034 D2534  ; #2腔体平移一级气缸伸出位延时设定值, #2腔体平移一级气缸伸出位感应延时[0002.02]
LD TR0
AND T1034  ; #2腔体平移一级气缸伸出位感应延时[0002.02]
OUT 802.02  ; #2腔体平移一级气缸伸出位标志[0002.02]

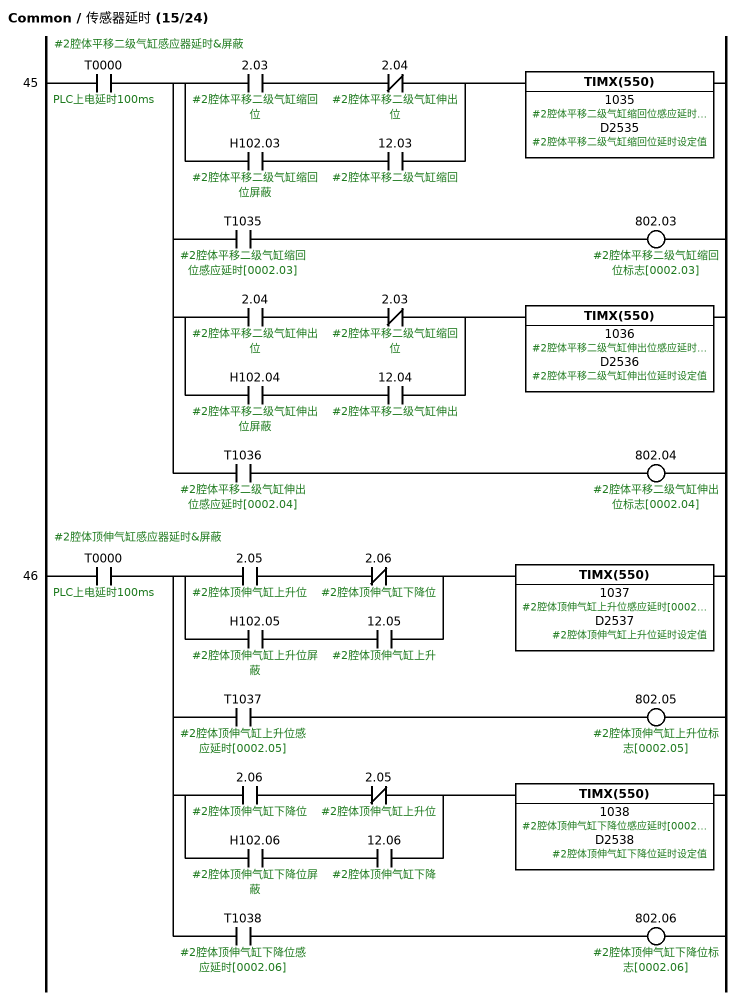
; rung 45: #2腔体平移二级气缸感应器延时&屏蔽
LD T0000  ; PLC上电延时100ms
OUT TR0
LD 2.03  ; #2腔体平移二级气缸缩回位
ANDNOT 2.04  ; #2腔体平移二级气缸伸出位
LD H102.03  ; #2腔体平移二级气缸缩回位屏蔽
AND 12.03  ; #2腔体平移二级气缸缩回
ORLD
ANDLD
TIMX(550) 1035 D2535  ; #2腔体平移二级气缸缩回位延时设定值, #2腔体平移二级气缸缩回位感应延时[0002.03]
LD TR0
AND T1035  ; #2腔体平移二级气缸缩回位感应延时[0002.03]
OUT 802.03  ; #2腔体平移二级气缸缩回位标志[0002.03]
LD TR0
LD 2.04  ; #2腔体平移二级气缸伸出位
ANDNOT 2.03  ; #2腔体平移二级气缸缩回位
LD H102.04  ; #2腔体平移二级气缸伸出位屏蔽
AND 12.04  ; #2腔体平移二级气缸伸出
ORLD
ANDLD
TIMX(550) 1036 D2536  ; #2腔体平移二级气缸伸出位延时设定值, #2腔体平移二级气缸伸出位感应延时[0002.04]
LD TR0
AND T1036  ; #2腔体平移二级气缸伸出位感应延时[0002.04]
OUT 802.04  ; #2腔体平移二级气缸伸出位标志[0002.04]
; rung 46: #2腔体顶伸气缸感应器延时&屏蔽
LD T0000  ; PLC上电延时100ms
OUT TR0
LD 2.05  ; #2腔体顶伸气缸上升位
ANDNOT 2.06  ; #2腔体顶伸气缸下降位
LD H102.05  ; #2腔体顶伸气缸上升位屏蔽
AND 12.05  ; #2腔体顶伸气缸上升
ORLD
ANDLD
TIMX(550) 1037 D2537  ; #2腔体顶伸气缸上升位延时设定值, #2腔体顶伸气缸上升位感应延时[0002.05]
LD TR0
AND T1037  ; #2腔体顶伸气缸上升位感应延时[0002.05]
OUT 802.05  ; #2腔体顶伸气缸上升位标志[0002.05]
LD TR0
LD 2.06  ; #2腔体顶伸气缸下降位
ANDNOT 2.05  ; #2腔体顶伸气缸上升位
LD H102.06  ; #2腔体顶伸气缸下降位屏蔽
AND 12.06  ; #2腔体顶伸气缸下降
ORLD
ANDLD
TIMX(550) 1038 D2538  ; #2腔体顶伸气缸下降位延时设定值, #2腔体顶伸气缸下降位感应延时[0002.06]
LD TR0
AND T1038  ; #2腔体顶伸气缸下降位感应延时[0002.06]
OUT 802.06  ; #2腔体顶伸气缸下降位标志[0002.06]

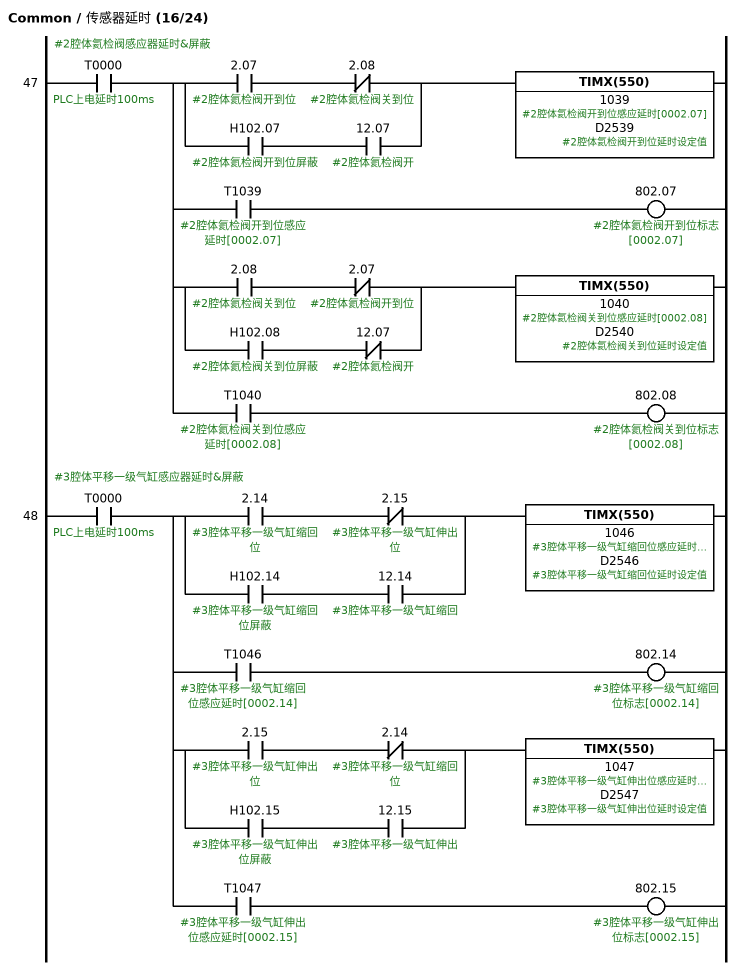
; rung 47: #2腔体氦检阀感应器延时&屏蔽
LD T0000  ; PLC上电延时100ms
OUT TR0
LD 2.07  ; #2腔体氦检阀开到位
ANDNOT 2.08  ; #2腔体氦检阀关到位
LD H102.07  ; #2腔体氦检阀开到位屏蔽
AND 12.07  ; #2腔体氦检阀开
ORLD
ANDLD
TIMX(550) 1039 D2539  ; #2腔体氦检阀开到位延时设定值, #2腔体氦检阀开到位感应延时[0002.07]
LD TR0
AND T1039  ; #2腔体氦检阀开到位感应延时[0002.07]
OUT 802.07  ; #2腔体氦检阀开到位标志[0002.07]
LD TR0
LD 2.08  ; #2腔体氦检阀关到位
ANDNOT 2.07  ; #2腔体氦检阀开到位
LD H102.08  ; #2腔体氦检阀关到位屏蔽
ANDNOT 12.07  ; #2腔体氦检阀开
ORLD
ANDLD
TIMX(550) 1040 D2540  ; #2腔体氦检阀关到位延时设定值, #2腔体氦检阀关到位感应延时[0002.08]
LD TR0
AND T1040  ; #2腔体氦检阀关到位感应延时[0002.08]
OUT 802.08  ; #2腔体氦检阀关到位标志[0002.08]
; rung 48: #3腔体平移一级气缸感应器延时&屏蔽
LD T0000  ; PLC上电延时100ms
OUT TR0
LD 2.14  ; #3腔体平移一级气缸缩回位
ANDNOT 2.15  ; #3腔体平移一级气缸伸出位
LD H102.14  ; #3腔体平移一级气缸缩回位屏蔽
AND 12.14  ; #3腔体平移一级气缸缩回
ORLD
ANDLD
TIMX(550) 1046 D2546  ; #3腔体平移一级气缸缩回位延时设定值, #3腔体平移一级气缸缩回位感应延时[0002.14]
LD TR0
AND T1046  ; #3腔体平移一级气缸缩回位感应延时[0002.14]
OUT 802.14  ; #3腔体平移一级气缸缩回位标志[0002.14]
LD TR0
LD 2.15  ; #3腔体平移一级气缸伸出位
ANDNOT 2.14  ; #3腔体平移一级气缸缩回位
LD H102.15  ; #3腔体平移一级气缸伸出位屏蔽
AND 12.15  ; #3腔体平移一级气缸伸出
ORLD
ANDLD
TIMX(550) 1047 D2547  ; #3腔体平移一级气缸伸出位延时设定值, #3腔体平移一级气缸伸出位感应延时[0002.15]
LD TR0
AND T1047  ; #3腔体平移一级气缸伸出位感应延时[0002.15]
OUT 802.15  ; #3腔体平移一级气缸伸出位标志[0002.15]

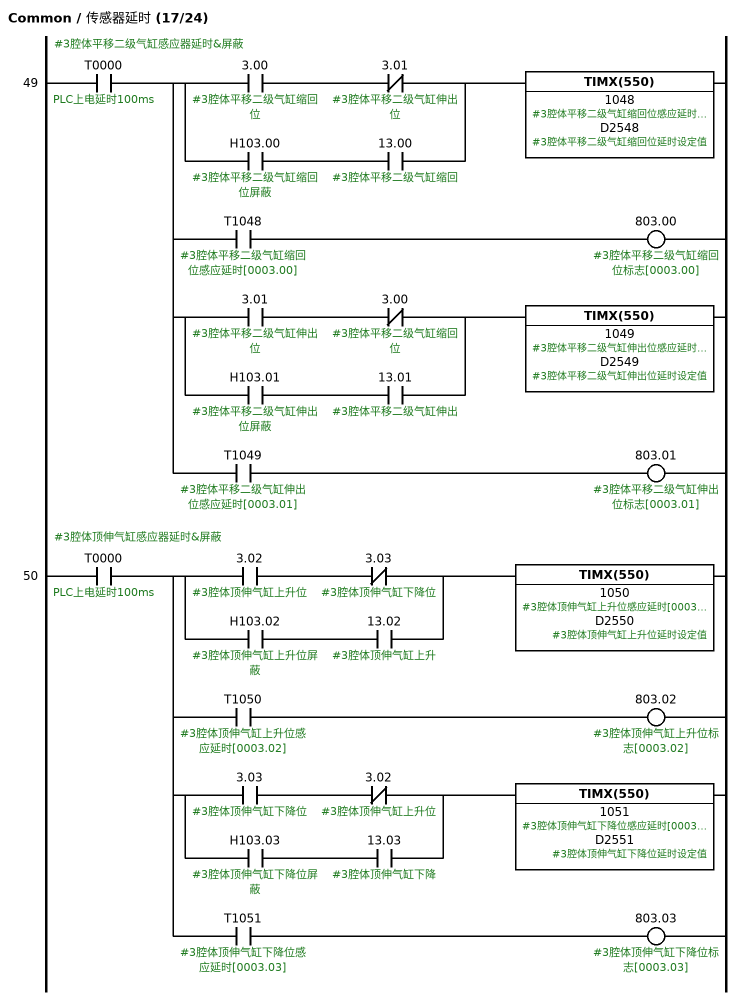
; rung 49: #3腔体平移二级气缸感应器延时&屏蔽
LD T0000  ; PLC上电延时100ms
OUT TR0
LD 3.00  ; #3腔体平移二级气缸缩回位
ANDNOT 3.01  ; #3腔体平移二级气缸伸出位
LD H103.00  ; #3腔体平移二级气缸缩回位屏蔽
AND 13.00  ; #3腔体平移二级气缸缩回
ORLD
ANDLD
TIMX(550) 1048 D2548  ; #3腔体平移二级气缸缩回位延时设定值, #3腔体平移二级气缸缩回位感应延时[0003.00]
LD TR0
AND T1048  ; #3腔体平移二级气缸缩回位感应延时[0003.00]
OUT 803.00  ; #3腔体平移二级气缸缩回位标志[0003.00]
LD TR0
LD 3.01  ; #3腔体平移二级气缸伸出位
ANDNOT 3.00  ; #3腔体平移二级气缸缩回位
LD H103.01  ; #3腔体平移二级气缸伸出位屏蔽
AND 13.01  ; #3腔体平移二级气缸伸出
ORLD
ANDLD
TIMX(550) 1049 D2549  ; #3腔体平移二级气缸伸出位延时设定值, #3腔体平移二级气缸伸出位感应延时[0003.01]
LD TR0
AND T1049  ; #3腔体平移二级气缸伸出位感应延时[0003.01]
OUT 803.01  ; #3腔体平移二级气缸伸出位标志[0003.01]
; rung 50: #3腔体顶伸气缸感应器延时&屏蔽
LD T0000  ; PLC上电延时100ms
OUT TR0
LD 3.02  ; #3腔体顶伸气缸上升位
ANDNOT 3.03  ; #3腔体顶伸气缸下降位
LD H103.02  ; #3腔体顶伸气缸上升位屏蔽
AND 13.02  ; #3腔体顶伸气缸上升
ORLD
ANDLD
TIMX(550) 1050 D2550  ; #3腔体顶伸气缸上升位延时设定值, #3腔体顶伸气缸上升位感应延时[0003.02]
LD TR0
AND T1050  ; #3腔体顶伸气缸上升位感应延时[0003.02]
OUT 803.02  ; #3腔体顶伸气缸上升位标志[0003.02]
LD TR0
LD 3.03  ; #3腔体顶伸气缸下降位
ANDNOT 3.02  ; #3腔体顶伸气缸上升位
LD H103.03  ; #3腔体顶伸气缸下降位屏蔽
AND 13.03  ; #3腔体顶伸气缸下降
ORLD
ANDLD
TIMX(550) 1051 D2551  ; #3腔体顶伸气缸下降位延时设定值, #3腔体顶伸气缸下降位感应延时[0003.03]
LD TR0
AND T1051  ; #3腔体顶伸气缸下降位感应延时[0003.03]
OUT 803.03  ; #3腔体顶伸气缸下降位标志[0003.03]

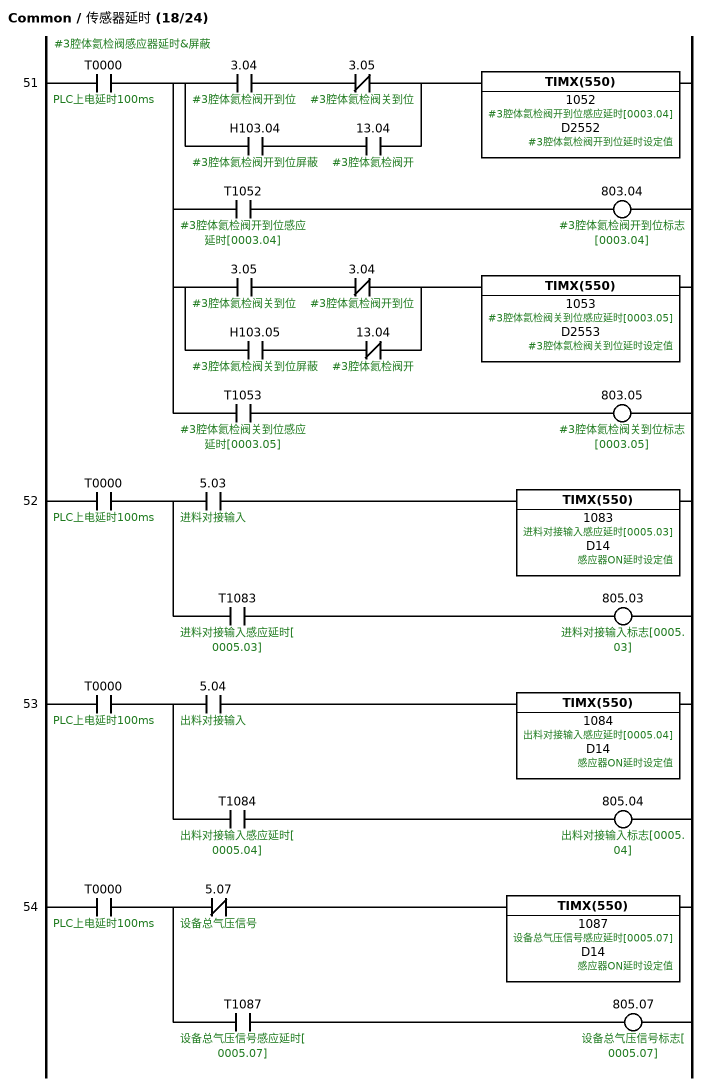
; rung 51: #3腔体氦检阀感应器延时&屏蔽
LD T0000  ; PLC上电延时100ms
OUT TR0
LD 3.04  ; #3腔体氦检阀开到位
ANDNOT 3.05  ; #3腔体氦检阀关到位
LD H103.04  ; #3腔体氦检阀开到位屏蔽
AND 13.04  ; #3腔体氦检阀开
ORLD
ANDLD
TIMX(550) 1052 D2552  ; #3腔体氦检阀开到位延时设定值, #3腔体氦检阀开到位感应延时[0003.04]
LD TR0
AND T1052  ; #3腔体氦检阀开到位感应延时[0003.04]
OUT 803.04  ; #3腔体氦检阀开到位标志[0003.04]
LD TR0
LD 3.05  ; #3腔体氦检阀关到位
ANDNOT 3.04  ; #3腔体氦检阀开到位
LD H103.05  ; #3腔体氦检阀关到位屏蔽
ANDNOT 13.04  ; #3腔体氦检阀开
ORLD
ANDLD
TIMX(550) 1053 D2553  ; #3腔体氦检阀关到位延时设定值, #3腔体氦检阀关到位感应延时[0003.05]
LD TR0
AND T1053  ; #3腔体氦检阀关到位感应延时[0003.05]
OUT 803.05  ; #3腔体氦检阀关到位标志[0003.05]
; rung 52
LD T0000  ; PLC上电延时100ms
OUT TR0
AND 5.03  ; 进料对接输入
TIMX(550) 1083 D14  ; 感应器ON延时设定值, 进料对接输入感应延时[0005.03]
LD TR0
AND T1083  ; 进料对接输入感应延时[0005.03]
OUT 805.03  ; 进料对接输入标志[0005.03]
; rung 53
LD T0000  ; PLC上电延时100ms
OUT TR0
AND 5.04  ; 出料对接输入
TIMX(550) 1084 D14  ; 感应器ON延时设定值, 出料对接输入感应延时[0005.04]
LD TR0
AND T1084  ; 出料对接输入感应延时[0005.04]
OUT 805.04  ; 出料对接输入标志[0005.04]
; rung 54
LD T0000  ; PLC上电延时100ms
OUT TR0
ANDNOT 5.07  ; 设备总气压信号
TIMX(550) 1087 D14  ; 感应器ON延时设定值, 设备总气压信号感应延时[0005.07]
LD TR0
AND T1087  ; 设备总气压信号感应延时[0005.07]
OUT 805.07  ; 设备总气压信号标志[0005.07]

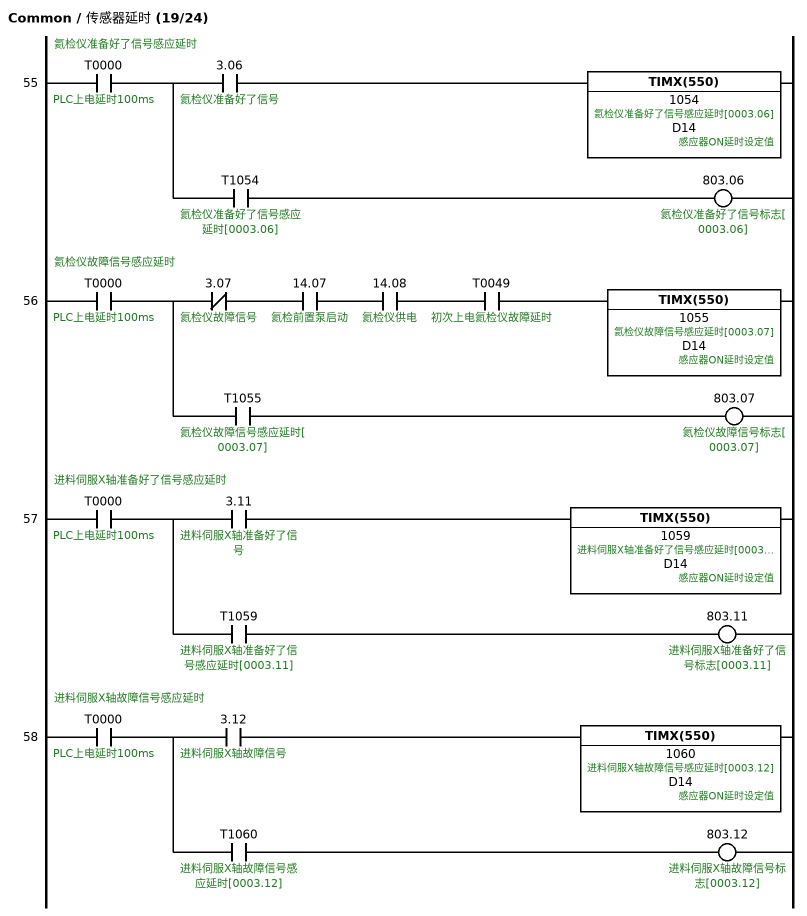
; rung 55: 氦检仪准备好了信号感应延时
LD T0000  ; PLC上电延时100ms
OUT TR0
AND 3.06  ; 氦检仪准备好了信号
TIMX(550) 1054 D14  ; 感应器ON延时设定值, 氦检仪准备好了信号感应延时[0003.06]
LD TR0
AND T1054  ; 氦检仪准备好了信号感应延时[0003.06]
OUT 803.06  ; 氦检仪准备好了信号标志[0003.06]
; rung 56: 氦检仪故障信号感应延时
LD T0000  ; PLC上电延时100ms
OUT TR0
ANDNOT 3.07  ; 氦检仪故障信号
AND 14.07  ; 氦检前置泵启动
AND 14.08  ; 氦检仪供电
AND T0049  ; 初次上电氦检仪故障延时
TIMX(550) 1055 D14  ; 感应器ON延时设定值, 氦检仪故障信号感应延时[0003.07]
LD TR0
AND T1055  ; 氦检仪故障信号感应延时[0003.07]
OUT 803.07  ; 氦检仪故障信号标志[0003.07]
; rung 57: 进料伺服X轴准备好了信号感应延时
LD T0000  ; PLC上电延时100ms
OUT TR0
AND 3.11  ; 进料伺服X轴准备好了信号
TIMX(550) 1059 D14  ; 感应器ON延时设定值, 进料伺服X轴准备好了信号感应延时[0003.11]
LD TR0
AND T1059  ; 进料伺服X轴准备好了信号感应延时[0003.11]
OUT 803.11  ; 进料伺服X轴准备好了信号标志[0003.11]
; rung 58: 进料伺服X轴故障信号感应延时
LD T0000  ; PLC上电延时100ms
OUT TR0
AND 3.12  ; 进料伺服X轴故障信号
TIMX(550) 1060 D14  ; 感应器ON延时设定值, 进料伺服X轴故障信号感应延时[0003.12]
LD TR0
AND T1060  ; 进料伺服X轴故障信号感应延时[0003.12]
OUT 803.12  ; 进料伺服X轴故障信号标志[0003.12]

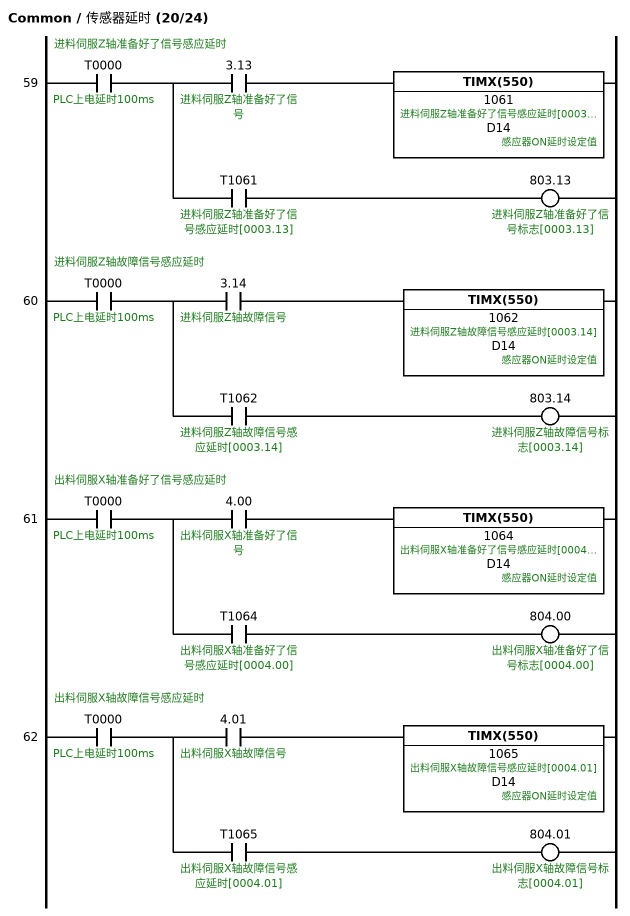
; rung 59: 进料伺服Z轴准备好了信号感应延时
LD T0000  ; PLC上电延时100ms
OUT TR0
AND 3.13  ; 进料伺服Z轴准备好了信号
TIMX(550) 1061 D14  ; 感应器ON延时设定值, 进料伺服Z轴准备好了信号感应延时[0003.13]
LD TR0
AND T1061  ; 进料伺服Z轴准备好了信号感应延时[0003.13]
OUT 803.13  ; 进料伺服Z轴准备好了信号标志[0003.13]
; rung 60: 进料伺服Z轴故障信号感应延时
LD T0000  ; PLC上电延时100ms
OUT TR0
AND 3.14  ; 进料伺服Z轴故障信号
TIMX(550) 1062 D14  ; 感应器ON延时设定值, 进料伺服Z轴故障信号感应延时[0003.14]
LD TR0
AND T1062  ; 进料伺服Z轴故障信号感应延时[0003.14]
OUT 803.14  ; 进料伺服Z轴故障信号标志[0003.14]
; rung 61: 出料伺服X轴准备好了信号感应延时
LD T0000  ; PLC上电延时100ms
OUT TR0
AND 4.00  ; 出料伺服X轴准备好了信号
TIMX(550) 1064 D14  ; 感应器ON延时设定值, 出料伺服X轴准备好了信号感应延时[0004.00]
LD TR0
AND T1064  ; 出料伺服X轴准备好了信号感应延时[0004.00]
OUT 804.00  ; 出料伺服X轴准备好了信号标志[0004.00]
; rung 62: 出料伺服X轴故障信号感应延时
LD T0000  ; PLC上电延时100ms
OUT TR0
AND 4.01  ; 出料伺服X轴故障信号
TIMX(550) 1065 D14  ; 感应器ON延时设定值, 出料伺服X轴故障信号感应延时[0004.01]
LD TR0
AND T1065  ; 出料伺服X轴故障信号感应延时[0004.01]
OUT 804.01  ; 出料伺服X轴故障信号标志[0004.01]

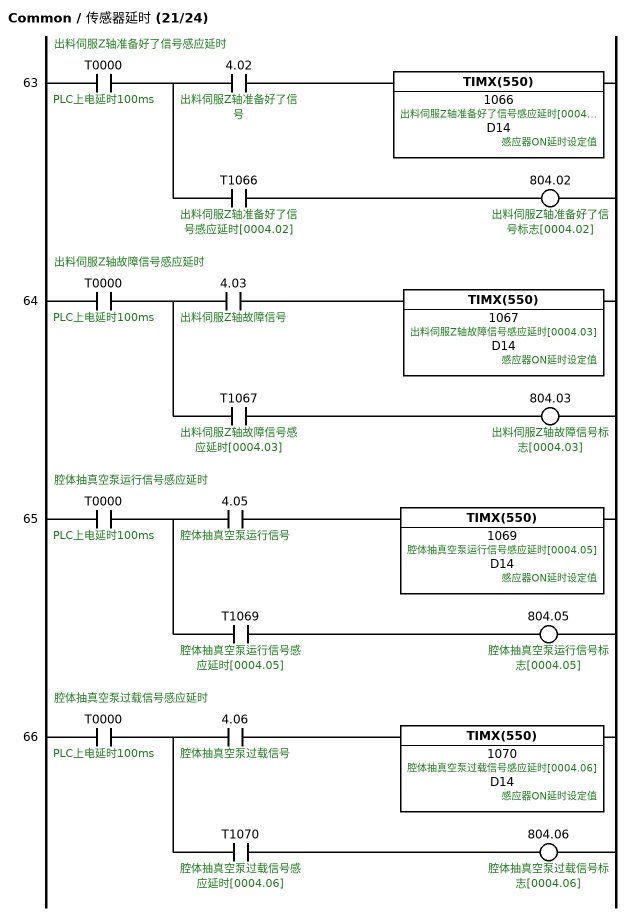
; rung 63: 出料伺服Z轴准备好了信号感应延时
LD T0000  ; PLC上电延时100ms
OUT TR0
AND 4.02  ; 出料伺服Z轴准备好了信号
TIMX(550) 1066 D14  ; 感应器ON延时设定值, 出料伺服Z轴准备好了信号感应延时[0004.02]
LD TR0
AND T1066  ; 出料伺服Z轴准备好了信号感应延时[0004.02]
OUT 804.02  ; 出料伺服Z轴准备好了信号标志[0004.02]
; rung 64: 出料伺服Z轴故障信号感应延时
LD T0000  ; PLC上电延时100ms
OUT TR0
AND 4.03  ; 出料伺服Z轴故障信号
TIMX(550) 1067 D14  ; 感应器ON延时设定值, 出料伺服Z轴故障信号感应延时[0004.03]
LD TR0
AND T1067  ; 出料伺服Z轴故障信号感应延时[0004.03]
OUT 804.03  ; 出料伺服Z轴故障信号标志[0004.03]
; rung 65: 腔体抽真空泵运行信号感应延时
LD T0000  ; PLC上电延时100ms
OUT TR0
AND 4.05  ; 腔体抽真空泵运行信号
TIMX(550) 1069 D14  ; 感应器ON延时设定值, 腔体抽真空泵运行信号感应延时[0004.05]
LD TR0
AND T1069  ; 腔体抽真空泵运行信号感应延时[0004.05]
OUT 804.05  ; 腔体抽真空泵运行信号标志[0004.05]
; rung 66: 腔体抽真空泵过载信号感应延时
LD T0000  ; PLC上电延时100ms
OUT TR0
AND 4.06  ; 腔体抽真空泵过载信号
TIMX(550) 1070 D14  ; 感应器ON延时设定值, 腔体抽真空泵过载信号感应延时[0004.06]
LD TR0
AND T1070  ; 腔体抽真空泵过载信号感应延时[0004.06]
OUT 804.06  ; 腔体抽真空泵过载信号标志[0004.06]

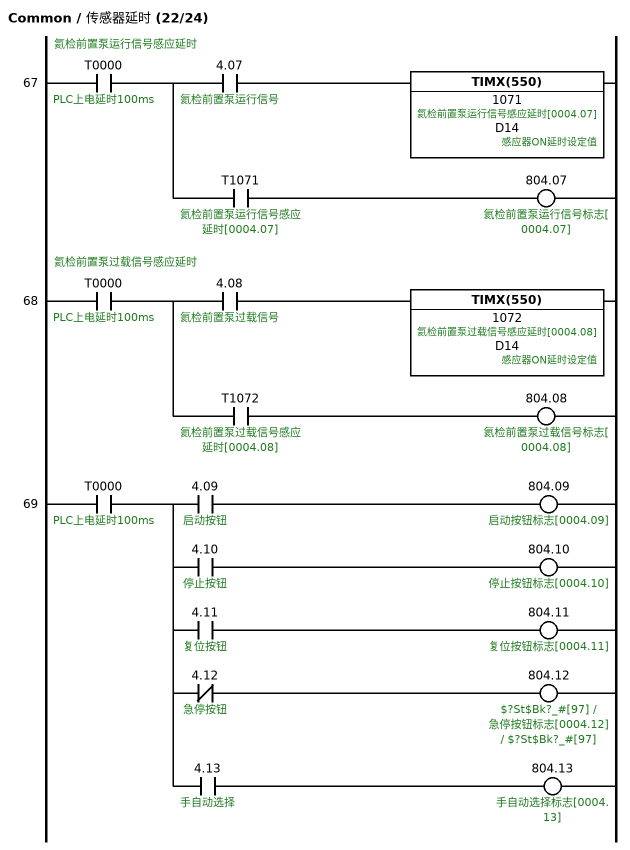
; rung 67: 氦检前置泵运行信号感应延时
LD T0000  ; PLC上电延时100ms
OUT TR0
AND 4.07  ; 氦检前置泵运行信号
TIMX(550) 1071 D14  ; 感应器ON延时设定值, 氦检前置泵运行信号感应延时[0004.07]
LD TR0
AND T1071  ; 氦检前置泵运行信号感应延时[0004.07]
OUT 804.07  ; 氦检前置泵运行信号标志[0004.07]
; rung 68: 氦检前置泵过载信号感应延时
LD T0000  ; PLC上电延时100ms
OUT TR0
AND 4.08  ; 氦检前置泵过载信号
TIMX(550) 1072 D14  ; 感应器ON延时设定值, 氦检前置泵过载信号感应延时[0004.08]
LD TR0
AND T1072  ; 氦检前置泵过载信号感应延时[0004.08]
OUT 804.08  ; 氦检前置泵过载信号标志[0004.08]
; rung 69
LD T0000  ; PLC上电延时100ms
OUT TR0
AND 4.09  ; 启动按钮
OUT 804.09  ; 启动按钮标志[0004.09]
LD TR0
AND 4.10  ; 停止按钮
OUT 804.10  ; 停止按钮标志[0004.10]
LD TR0
AND 4.11  ; 复位按钮
OUT 804.11  ; 复位按钮标志[0004.11]
LD TR0
ANDNOT 4.12  ; 急停按钮
OUT 804.12  ; $?St$Bk?_#[97] / 急停按钮标志[0004.12] / $?St$Bk?_#[97]
LD TR0
AND 4.13  ; 手自动选择
OUT 804.13  ; 手自动选择标志[0004.13]

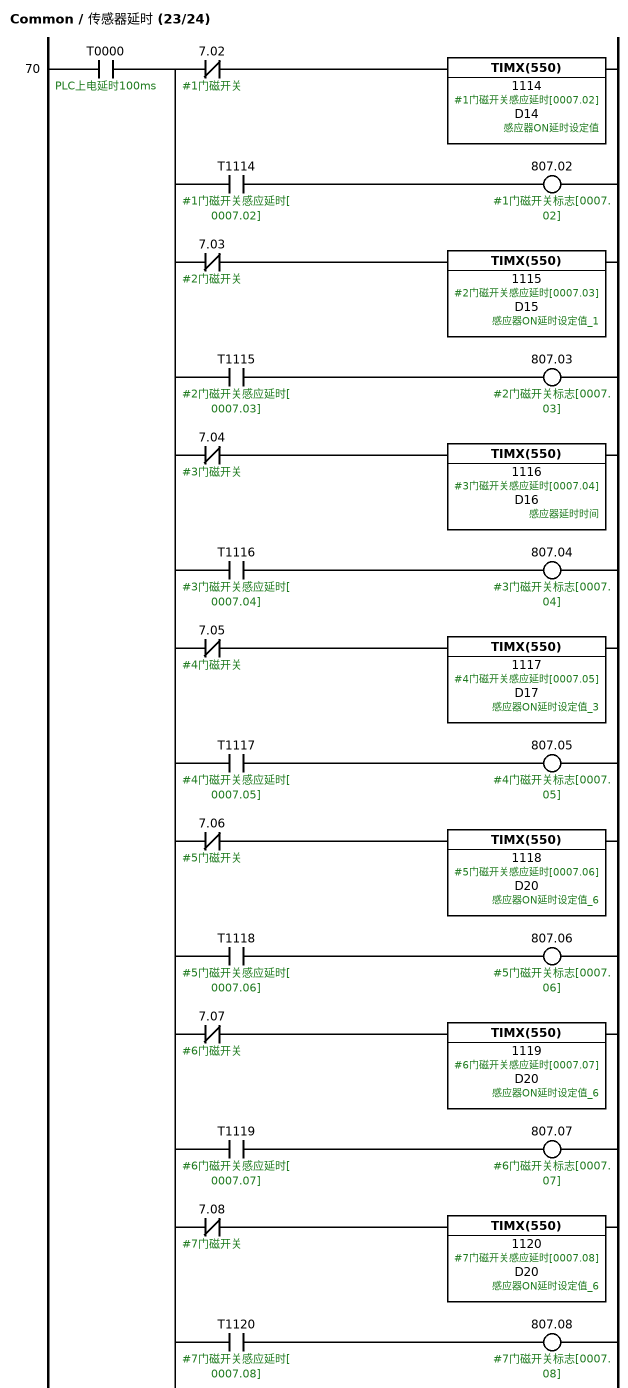

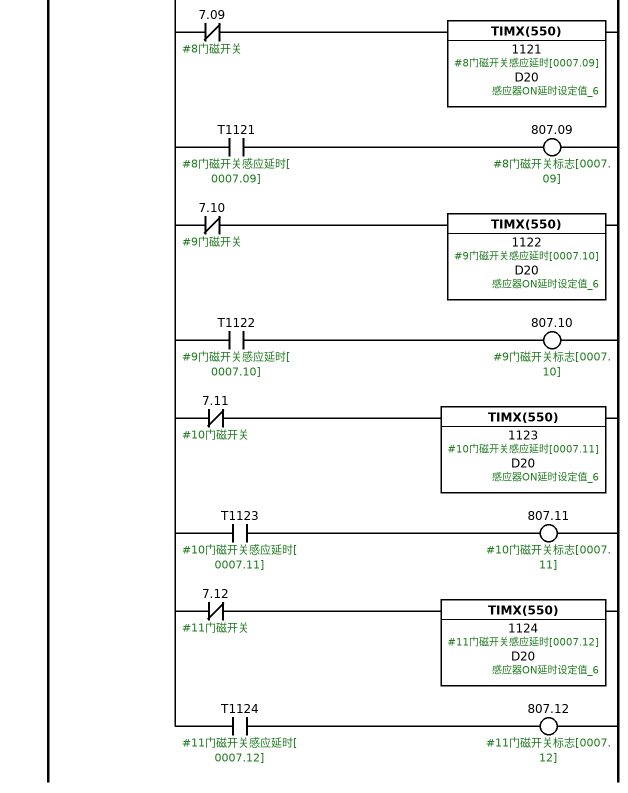
; rung 70
LD T0000  ; PLC上电延时100ms
OUT TR0
ANDNOT 7.02  ; #1门磁开关
TIMX(550) 1114 D14  ; 感应器ON延时设定值, #1门磁开关感应延时[0007.02]
LD TR0
AND T1114  ; #1门磁开关感应延时[0007.02]
OUT 807.02  ; #1门磁开关标志[0007.02]
LD TR0
ANDNOT 7.03  ; #2门磁开关
TIMX(550) 1115 D15  ; 感应器ON延时设定值_1, #2门磁开关感应延时[0007.03]
LD TR0
AND T1115  ; #2门磁开关感应延时[0007.03]
OUT 807.03  ; #2门磁开关标志[0007.03]
LD TR0
ANDNOT 7.04  ; #3门磁开关
TIMX(550) 1116 D16  ; 感应器延时时间, #3门磁开关感应延时[0007.04]
LD TR0
AND T1116  ; #3门磁开关感应延时[0007.04]
OUT 807.04  ; #3门磁开关标志[0007.04]
LD TR0
ANDNOT 7.05  ; #4门磁开关
TIMX(550) 1117 D17  ; 感应器ON延时设定值_3, #4门磁开关感应延时[0007.05]
LD TR0
AND T1117  ; #4门磁开关感应延时[0007.05]
OUT 807.05  ; #4门磁开关标志[0007.05]
LD TR0
ANDNOT 7.06  ; #5门磁开关
TIMX(550) 1118 D20  ; 感应器ON延时设定值_6, #5门磁开关感应延时[0007.06]
LD TR0
AND T1118  ; #5门磁开关感应延时[0007.06]
OUT 807.06  ; #5门磁开关标志[0007.06]
LD TR0
ANDNOT 7.07  ; #6门磁开关
TIMX(550) 1119 D20  ; 感应器ON延时设定值_6, #6门磁开关感应延时[0007.07]
LD TR0
AND T1119  ; #6门磁开关感应延时[0007.07]
OUT 807.07  ; #6门磁开关标志[0007.07]
LD TR0
ANDNOT 7.08  ; #7门磁开关
TIMX(550) 1120 D20  ; 感应器ON延时设定值_6, #7门磁开关感应延时[0007.08]
LD TR0
AND T1120  ; #7门磁开关感应延时[0007.08]
OUT 807.08  ; #7门磁开关标志[0007.08]
LD TR0
ANDNOT 7.09  ; #8门磁开关
TIMX(550) 1121 D20  ; 感应器ON延时设定值_6, #8门磁开关感应延时[0007.09]
LD TR0
AND T1121  ; #8门磁开关感应延时[0007.09]
OUT 807.09  ; #8门磁开关标志[0007.09]
LD TR0
ANDNOT 7.10  ; #9门磁开关
TIMX(550) 1122 D20  ; 感应器ON延时设定值_6, #9门磁开关感应延时[0007.10]
LD TR0
AND T1122  ; #9门磁开关感应延时[0007.10]
OUT 807.10  ; #9门磁开关标志[0007.10]
LD TR0
ANDNOT 7.11  ; #10门磁开关
TIMX(550) 1123 D20  ; 感应器ON延时设定值_6, #10门磁开关感应延时[0007.11]
LD TR0
AND T1123  ; #10门磁开关感应延时[0007.11]
OUT 807.11  ; #10门磁开关标志[0007.11]
LD TR0
ANDNOT 7.12  ; #11门磁开关
TIMX(550) 1124 D20  ; 感应器ON延时设定值_6, #11门磁开关感应延时[0007.12]
LD TR0
AND T1124  ; #11门磁开关感应延时[0007.12]
OUT 807.12  ; #11门磁开关标志[0007.12]

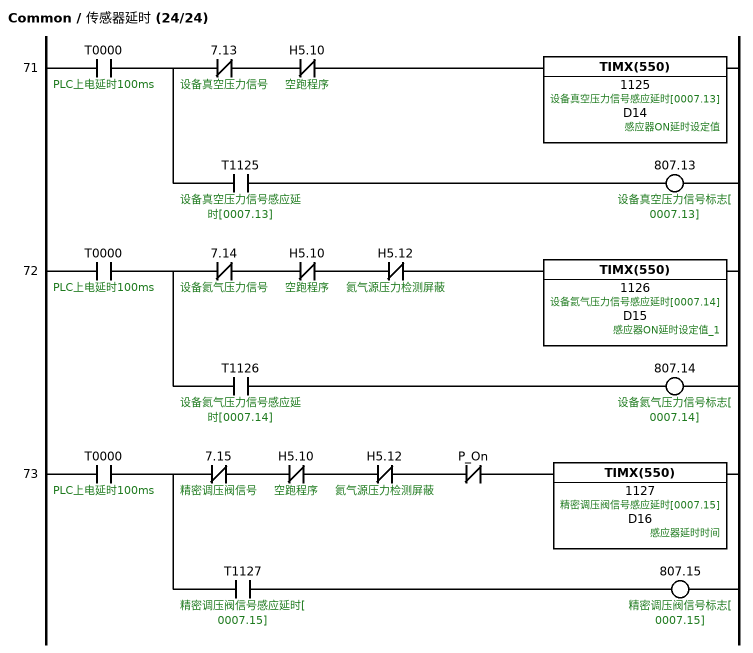
; rung 71
LD T0000  ; PLC上电延时100ms
OUT TR0
ANDNOT 7.13  ; 设备真空压力信号
ANDNOT H5.10  ; 空跑程序
TIMX(550) 1125 D14  ; 感应器ON延时设定值, 设备真空压力信号感应延时[0007.13]
LD TR0
AND T1125  ; 设备真空压力信号感应延时[0007.13]
OUT 807.13  ; 设备真空压力信号标志[0007.13]
; rung 72
LD T0000  ; PLC上电延时100ms
OUT TR0
ANDNOT 7.14  ; 设备氦气压力信号
ANDNOT H5.10  ; 空跑程序
ANDNOT H5.12  ; 氦气源压力检测屏蔽
TIMX(550) 1126 D15  ; 感应器ON延时设定值_1, 设备氦气压力信号感应延时[0007.14]
LD TR0
AND T1126  ; 设备氦气压力信号感应延时[0007.14]
OUT 807.14  ; 设备氦气压力信号标志[0007.14]
; rung 73
LD T0000  ; PLC上电延时100ms
OUT TR0
ANDNOT 7.15  ; 精密调压阀信号
ANDNOT H5.10  ; 空跑程序
ANDNOT H5.12  ; 氦气源压力检测屏蔽
ANDNOT P_On
TIMX(550) 1127 D16  ; 感应器延时时间, 精密调压阀信号感应延时[0007.15]
LD TR0
AND T1127  ; 精密调压阀信号感应延时[0007.15]
OUT 807.15  ; 精密调压阀信号标志[0007.15]

### Section 数据传递

